			ARDs4StepUpDownMovement[iPull4StepFL].lrZone1Acc						:= fbA31ArmSpeedProfileMemory.ARDsArmSpeedProfileMemory[fbA21UpDownPattern.ARDsUpdownPatternMemory[ARi4StepPatternNo[iPull4StepFL]].iZone1SpdProfileNo].lrAcc;
			ARDs4StepUpDownMovement[iPull4StepFL].lrZone1Dcc						:= fbA31ArmSpeedProfileMemory.ARDsArmSpeedProfileMemory[fbA21UpDownPattern.ARDsUpdownPatternMemory[ARi4StepPatternNo[iPull4StepFL]].iZone1SpdProfileNo].lrDcc;
			ARDs4StepUpDownMovement[iPull4StepFL].lrZone2Acc						:= fbA31ArmSpeedProfileMemory.ARDsArmSpeedProfileMemory[fbA21UpDownPattern.ARDsUpdownPatternMemory[ARi4StepPatternNo[iPull4StepFL]].iZone2SpdProfileNo].lrAcc;
			ARDs4StepUpDownMovement[iPull4StepFL].lrZone2Dcc						:= fbA31ArmSpeedProfileMemory.ARDsArmSpeedProfileMemory[fbA21UpDownPattern.ARDsUpdownPatternMemory[ARi4StepPatternNo[iPull4StepFL]].iZone2SpdProfileNo].lrDcc;
			ARDs4StepUpDownMovement[iPull4StepFL].lrZone3Acc						:= fbA31ArmSpeedProfileMemory.ARDsArmSpeedProfileMemory[fbA21UpDownPattern.ARDsUpdownPatternMemory[ARi4StepPatternNo[iPull4StepFL]].iZone3SpdProfileNo].lrAcc;
			ARDs4StepUpDownMovement[iPull4StepFL].lrZone3Dcc						:= fbA31ArmSpeedProfileMemory.ARDsArmSpeedProfileMemory[fbA21UpDownPattern.ARDsUpdownPatternMemory[ARi4StepPatternNo[iPull4StepFL]].iZone3SpdProfileNo].lrDcc;
			ARDs4StepUpDownMovement[iPull4StepFL].lrZone4Acc						:= fbA31ArmSpeedProfileMemory.ARDsArmSpeedProfileMemory[fbA21UpDownPattern.ARDsUpdownPatternMemory[ARi4StepPatternNo[iPull4StepFL]].iZone4SpdProfileNo].lrAcc;
			ARDs4StepUpDownMovement[iPull4StepFL].lrZone4Dcc						:= fbA31ArmSpeedProfileMemory.ARDsArmSpeedProfileMemory[fbA21UpDownPattern.ARDsUpdownPatternMemory[ARi4StepPatternNo[iPull4StepFL]].iZone4SpdProfileNo].lrDcc;

			ARDs4StepUpDownMovement[iPull4StepFL].sReservedLreal;
			ARDs4StepUpDownMovement[iPull4StepFL].sUpDownPatternDescription	:= fbA21UpDownPattern.ARDsUpdownPatternMemory[ARi4StepPatternNo[iPull4StepFL]].sDescription;
	END_IF
END_FOR

(*[][][][][][][][][][][][][][][][][][][][][][][][][][][][][][][][][][][][][][][][][][][][][][][][][][][][][][][][][][][][][][][][][][][][][][][][][][][][][][][][][][][][][][][][][][][][][][][][][][][]*)
(*Check Which Staton Request for Data*)
iCallCheck := 0;
bCalledDataRequestStationFound := FALSE;

FOR iCallCheck := 0 TO iStnQty DO
		IF ARbProductRecipeCallEn[iCallCheck] THEN
		iCalledDataRequestFromStationNo := iCallCheck;
		bCalledDataRequestStationFound := TRUE;
		iCallCheck := 28;
		END_IF
END_FOR

IF NOT bCalledDataRequestStationFound AND iCallCheck < iStnQty THEN
		iCalledDataRequestFromStationNo := 0;
END_IF

iProductRecipeNoCall := ARiProductRecipeNoCall[iCalledDataRequestFromStationNo];
iProductRecipeStepCall := ARiProductRecipeStepCall[iCalledDataRequestFromStationNo];
bCallSt := bCalledDataRequestStationFound;


(*[][][][][][][][][][][][][][][][][][][][][][][][][][][][][][][][][][][][][][][][][][][][][][][][][][][][][][][][][][][][][][][][][][][][][][][][][][][][][][][][][][][][][][][][][][][][][][][][][][][]*)
(*Reset fb*)
bCallStRE(CLK:=bCallSt , Q=> );
bCallStFE(CLK:=bCallSt , Q=> );

IF bCallStRE.Q OR bCallStFE.Q THEN
DSA1fbPnpSequenceMemoryCall.bCallPB := FALSE;
DSA21UpDownPatternCall.bCallPB := FALSE;
DSA31ArmSpeedProfileCall.bCallPB := FALSE;
DSfbGnrProductRecipeMemoryOut.bCallCompleted := FALSE;
DSfbGnrProductRecipeMemoryOut.bCallArmSpeedProfileMemoryErr := FALSE;
DSfbGnrProductRecipeMemoryOut.bCallUpDownPatternMemoryErr := FALSE;
DSfbGnrProductRecipeMemoryOut.bCallPickStationNoErr := FALSE;
DSfbGnrProductRecipeMemoryOut.bCallTransferStationNoErr := FALSE;

iBufferPickStationNo:= 0;
iBufferTransferStationNo:= 0;
iBufferDownPickPatternNo:= 0;
iBufferUpPickPatternNo:= 0;
iBufferDownTransferPatternNo:= 0;
iBufferUpTransferPatternNo:= 0;
(*
DSfbGnrProductRecipeMemoryOut.DSGnrCalledArmPnpParameter.iCallArmNo := 0;
DSfbGnrProductRecipeMemoryOut.DSGnrCalledArmPnpParameter.iPickStationNo := 0;
DSfbGnrProductRecipeMemoryOut.DSGnrCalledArmPnpParameter.iTransferStationNo := 0;
*)
DSfbGnrProductRecipeMemoryOut.iCallCaseNo := 0;

END_IF
(*
(*Limit Loading and Unloading ID*)
IF ARiLdStnID < iStnQty THEN
ARiLdStnID:= iStnQty + 1;
END_IF
IF ARiUldStnID < iStnQty THEN
ARiUldStnID:= iStnQty + 2;
END_IF
*)


(*Reset Err after 0.5Sec*)
(*
tCallPickStationNoErrTimer(IN:= DSfbGnrProductRecipeMemoryOut.bCallPickStationNoErr , PT:=t#0.5s , Q=> , ET=> );
*)
IF tCallPickStationNoErrTimer.Q OR NOT bCallSt THEN
DSfbGnrProductRecipeMemoryOut.bCallPickStationNoErr := FALSE;
END_IF

(*
tCallTransferStationNoErrTimer(IN:= DSfbGnrProductRecipeMemoryOut.bCallTransferStationNoErr , PT:=t#0.5s , Q=> , ET=> );
*)
IF tCallTransferStationNoErrTimer.Q OR NOT bCallSt THEN
DSfbGnrProductRecipeMemoryOut.bCallTransferStationNoErr := FALSE;
END_IF

(*
tCallArmSpeedProfileMemoryErrTimer(IN:= DSfbGnrProductRecipeMemoryOut.bCallArmSpeedProfileMemoryErr , PT:=t#0.5s , Q=> , ET=> );
*)
IF tCallArmSpeedProfileMemoryErrTimer.Q OR NOT bCallSt THEN
DSfbGnrProductRecipeMemoryOut.bCallArmSpeedProfileMemoryErr := FALSE;
END_IF

(*
tCallUpDownPatternMemoryErrTimer(IN:= DSfbGnrProductRecipeMemoryOut.bCallUpDownPatternMemoryErr , PT:=t#0.5s , Q=> , ET=> );
*)
IF tCallUpDownPatternMemoryErrTimer.Q OR NOT bCallSt THEN
DSfbGnrProductRecipeMemoryOut.bCallUpDownPatternMemoryErr := FALSE;
END_IF

(*Trigger Error*)

IF (iProductRecipeNoCall <= 0 OR iProductRecipeNoCall > iProductRecipeArrayQty) AND bCallSt THEN
DSfbGnrProductRecipeMemoryOut.bInvalidProductRecipeNoErrHold := TRUE;
ELSE
DSfbGnrProductRecipeMemoryOut.bInvalidProductRecipeNoErrHold := FALSE;
END_IF

IF (iProductRecipeStepCall <= 0 OR iProductRecipeStepCall > iProductRecipeStepArrayQty) AND bCallSt THEN
DSfbGnrProductRecipeMemoryOut.bInvalidProductRecipeStepErrHold := TRUE;
ELSE
DSfbGnrProductRecipeMemoryOut.bInvalidProductRecipeStepErrHold := FALSE;
END_IF

rebInvalidProductRecipeNo(CLK:=DSfbGnrProductRecipeMemoryOut.bInvalidProductRecipeNoErrHold AND bCallSt , Q=> );

IF rebInvalidProductRecipeNo.Q THEN
DSfbGnrProductRecipeMemoryOut.bInvalidProductRecipeNoErrPulse := TRUE;
END_IF

rebInvalidProductRecipeStep(CLK:=DSfbGnrProductRecipeMemoryOut.bInvalidProductRecipeStepErrHold AND bCallSt , Q=> );

IF rebInvalidProductRecipeStep.Q THEN
DSfbGnrProductRecipeMemoryOut.bInvalidProductRecipeStepErrPulse := TRUE;
END_IF


tInvalidProductRecipeNoErrTimer(IN:= DSfbGnrProductRecipeMemoryOut.bInvalidProductRecipeNoErrHold , PT:=t#0.5s , Q=> , ET=> );

IF tInvalidProductRecipeNoErrTimer.Q OR NOT bCallSt THEN
DSfbGnrProductRecipeMemoryOut.bInvalidProductRecipeNoErrPulse := FALSE;
END_IF


tInvalidProductRecipeStepErrTimer(IN:= DSfbGnrProductRecipeMemoryOut.bInvalidProductRecipeStepErrHold , PT:=t#0.5s , Q=> , ET=> );

IF tInvalidProductRecipeStepErrTimer.Q OR NOT bCallSt THEN
DSfbGnrProductRecipeMemoryOut.bInvalidProductRecipeStepErrPulse := FALSE;
END_IF

(*Declare FB*)

fbA1PnpSequenceMemory(
	bSavePB:=bSavePB ,
	bLoadPB:= bLoadPB,
	bClearPB:=bClearPB,
	bCopyPB:=DSA1fbPnpSequenceMemoryStore.bCopyPB ,
	iCopyToProductRecipeNo:=DSA1fbPnpSequenceMemoryStore.iCopyToProductRecipeNo ,
(*	ARiLdStnID:= ARiLdStnID,
	ARiUldStnID:= ARiUldStnID,
*)	iProductRecipeNo:=DSA1fbPnpSequenceMemoryStore.iProductRecipeNo ,
	DSA1inPnpSequenceMemory:=DSA1fbPnpSequenceMemoryStore.DsA1inPnpSequenceMemory ,
	Call_iProductRecipeNo:=DSA1fbPnpSequenceMemoryCall.Call_iProductRecipeNo ,
	bCallPB:=DSA1fbPnpSequenceMemoryCall.bCallPB ,
	bSaveInd=>bSaveInd ,
	bLoadInd=> bLoadInd,
	bClearInd=>bClearInd,
	bCallCompleted=>DSA1fbPnpSequenceMemoryCall.bCallCompleted ,
	bInvalidCallProductRecipeNoHold=>DSA1fbPnpSequenceMemoryCall.bInvalidCallProductRecipeNoHold ,
	bInvalidCallProductRecipeNoPulse=>DSA1fbPnpSequenceMemoryCall.bInvalidCallProductRecipeNoPulse ,
	Call_DSA1PnpSequenceMemory=>DSA1fbPnpSequenceMemoryCall.Call_DsPnpSequenceMemory );

fbA21UpDownPattern(
	bSavePB:=bSavePB ,
	bLoadPB:= bLoadPB,
	bCopyPB:=DSA21UpDownPatternStore.bCopyPB ,
	iCopyToUpDownPatternNo:= DSA21UpDownPatternStore.iCopyToUpDownPatternNo,
	iUpDownPatternNo:=DSA21UpDownPatternStore.iUpDownPatternNo ,
	DSinUpDownPatternMemory:=DSA21UpDownPatternStore.DsInUpDownPatternMemory ,
	Call_iUpDownPatternNo:=DSA21UpDownPatternCall.Call_iUpDownPatternNo ,
	bCallPB:=DSA21UpDownPatternCall.bCallPB ,
	bSaveInd=>bSaveInd ,
	bLoadInd=>bLoadInd,
	bCallCompleted=>DSA21UpDownPatternCall.bCallCompleted ,
	bInvalidCallUpdownPatternNoHold=>DSA21UpDownPatternCall.bInvalidCallUpDownPatternNoHold ,
	bInvalidCallUpdownPatternNoPulse=>DSA21UpDownPatternCall.bInvalidCallUpDownPatternNoPulse ,
	Call_DSUpdownPattern=>DSA21UpDownPatternCall.Call_DsUpDownPattern );

fbA31ArmSpeedProfileMemory(
	bSavePB:= bSavePB,
	bLoadPB:= bLoadPB,
	bCopyPB:=DSA31ArmSpeedProfileStore.bCopyPB ,
	iCopyToSpdProfileNo:=DSA31ArmSpeedProfileStore.iCopyToSpdProfileNo ,
	iVertMaxVelo:=iVertMaxVelo ,
	iVertMaxAcc:=iVertMaxAcc ,
	iVertMaxDcc:=iVertMaxDcc ,
	iVertMinVelo:=iVertMinVelo ,
	iVertMinAcc:=iVertMinAcc ,
	iVertMinDcc:=iVertMinDcc ,
	iArmSpdProfileNo:= DSA31ArmSpeedProfileStore.iArmSpdProfileNo,
	DSArmSpeedProfile:= DSA31ArmSpeedProfileStore.DsArmSpeedProfile,
	Call_iArmSpdProfile:= DSA31ArmSpeedProfileCall.Call_iArmSpdProfile ,
	bCallPB:= DSA31ArmSpeedProfileCall.bCallPB ,
	bSaveInd=>bSaveInd ,
	bLoadInd=>bLoadInd ,
	bCallCompleted=>DSA31ArmSpeedProfileCall.bCallCompleted ,
	bInvalidCallArmSpdProfileNoHold=> DSA31ArmSpeedProfileCall.bInvalidCallArmSpdProfileNoHold,
	bInvalidCallArmSpdProfileNoPulse=> DSA31ArmSpeedProfileCall.bInvalidCallArmSpdProfileNoPulse,
	Call_DSArmSpeedProfile=>DSA31ArmSpeedProfileCall.Call_DSArmSpdProfile );

fbV2A32MachineZoneHeight(
	ARDSLdZoneHeight:=ARDSLdZoneHeight ,
	ARDSStationZoneHeight:=ARDSStationZoneHeight ,
	ARDSUldZoneHeight:=ARDSUldZoneHeight ,
	ARDSLdZonePosOut=>ARDSLdZonePosOut ,
	ARDSStationZonePosOut=>ARDSStationZonePosOut ,
	ARDSUldZonePosOut=>ARDSUldZonePosOut );



(*Call Start*)

rebCallSt(CLK:=bCallSt , Q=> );
IF rebCallSt.Q AND NOT DSfbGnrProductRecipeMemoryOut.bInvalidProductRecipeNoErrHold AND NOT DSfbGnrProductRecipeMemoryOut.bInvalidProductRecipeStepErrHold(*) OR febInvalidProcessStep.Q*) THEN
DSfbGnrProductRecipeMemoryOut.iCallCaseNo := 1;
END_IF



rebInvalidUpDownPatternMemoryCall(CLK:=DSA21UpDownPatternCall.bInvalidCallUpDownPatternNoHold , Q=> );
rebInvalidSpeedProfileMemoryCall(CLK:=DSA31ArmSpeedProfileCall.bInvalidCallArmSpdProfileNoHold , Q=> );



CASE DSfbGnrProductRecipeMemoryOut.iCallCaseNo OF

0:;

1: (*Select PnpSequenceNo By Refering iProductRecipeNoCall*)
DSfbGnrProductRecipeMemoryOut.bCallUpDownPatternMemoryErr := FALSE;
DSfbGnrProductRecipeMemoryOut.bCallArmSpeedProfileMemoryErr := FALSE;
DSfbGnrProductRecipeMemoryOut.bCallPickStationNoErr := FALSE;
DSfbGnrProductRecipeMemoryOut.bCallTransferStationNoErr := FALSE;


DSA1fbPnpSequenceMemoryCall.Call_iProductRecipeNo := iProductRecipeNoCall;
DSA1fbPnpSequenceMemoryCall.bCallPB := TRUE;
DSfbGnrProductRecipeMemoryOut.iCalledProductRecipeNo := iProductRecipeNoCall;
DSfbGnrProductRecipeMemoryOut.iCalledProductRecipeStep := iProductRecipeStepCall;

IF DSA1fbPnpSequenceMemoryCall.bCallCompleted THEN
DSA1fbPnpSequenceMemoryCall.bCallPB := FALSE;



DSfbGnrProductRecipeMemoryOut.iCallCaseNo:=10;

END_IF


(*[][][][][][][][][][][][][][][][][][][][][][][][][][][][][][][][][][][][][][][][][][][][][][][][][][][][][][][][][][][][][][][][][][][][][][][][][][][][][][][][][][][][][][][][][][][][][][][][][][][]*)
62: (* Feed Transfer Station Vertical Zone Position*)


DSfbGnrProductRecipeMemoryOut.DSGnrCalledArmPnpParameter.iTransferStationNo := iBufferTransferStationNo;

iTransLdStnID := 0;
iTransUldStnID := 0;
bTransLdStnFound := FALSE;
bTransUldStnFound := FALSE;

iBufTransStnNoCheckFL := 1;
	FOR iBufTransStnNoCheckFL := 1 TO iLdStnQty DO
		IF iBufTransStnNoCheckFL >=1 AND iBufTransStnNoCheckFL <= iLdStnQty THEN
			IF iBufferTransferStationNo = ARiLdStnID[iBufTransStnNoCheckFL] THEN
				iTransLdStnID := iBufTransStnNoCheckFL;
				bTransLdStnFound := TRUE;
				iBufTransStnNoCheckFL := iLdStnQty +2;
			END_IF
		END_IF
	END_FOR

iBufTransStnNoCheckFL := 1;
	FOR iBufTransStnNoCheckFL := 1 TO iUldStnQty DO
		IF iBufTransStnNoCheckFL >=1 AND iBufTransStnNoCheckFL <= iUldStnQty THEN
			IF iBufferTransferStationNo = ARiUldStnID[iBufTransStnNoCheckFL] THEN
				iTransUldStnID := iBufTransStnNoCheckFL;
				bTransUldStnFound := TRUE;
				iBufTransStnNoCheckFL := iUldStnQty +2;
			END_IF
		END_IF
	END_FOR


IF bTransLdStnFound THEN

		IF bEnableCallArmNo THEN
			DSfbGnrProductRecipeMemoryOut.DSGnrCalledArmPnpParameter.DSA1DownTransferMovement.lrZone1StartPos := ARDSLdZonePosOut[iTransLdStnID].lrZone1StartPos - ARiVertArmPosOffset[iCallArmNo] ;
			DSfbGnrProductRecipeMemoryOut.DSGnrCalledArmPnpParameter.DSA1DownTransferMovement.lrZone2StartPos := ARDSLdZonePosOut[iTransLdStnID].lrZone2StartPos - ARiVertArmPosOffset[iCallArmNo] ;
			DSfbGnrProductRecipeMemoryOut.DSGnrCalledArmPnpParameter.DSA1DownTransferMovement.lrZone3StartPos := ARDSLdZonePosOut[iTransLdStnID].lrZone3StartPos - ARiVertArmPosOffset[iCallArmNo] ;
			DSfbGnrProductRecipeMemoryOut.DSGnrCalledArmPnpParameter.DSA1DownTransferMovement.lrZone4StartPos := ARDSLdZonePosOut[iTransLdStnID].lrZone4StartPos - ARiVertArmPosOffset[iCallArmNo] ;

			DSfbGnrProductRecipeMemoryOut.DSGnrCalledArmPnpParameter.DSA1DownTransferMovement.lrZone1EndPos := ARDSLdZonePosOut[iTransLdStnID].lrZone1EndPos - ARiVertArmPosOffset[iCallArmNo] ;
			DSfbGnrProductRecipeMemoryOut.DSGnrCalledArmPnpParameter.DSA1DownTransferMovement.lrZone2EndPos := ARDSLdZonePosOut[iTransLdStnID].lrZone2EndPos - ARiVertArmPosOffset[iCallArmNo] ;
			DSfbGnrProductRecipeMemoryOut.DSGnrCalledArmPnpParameter.DSA1DownTransferMovement.lrZone3EndPos := ARDSLdZonePosOut[iTransLdStnID].lrZone3EndPos - ARiVertArmPosOffset[iCallArmNo] ;
			DSfbGnrProductRecipeMemoryOut.DSGnrCalledArmPnpParameter.DSA1DownTransferMovement.lrZone4EndPos := ARDSLdZonePosOut[iTransLdStnID].lrZone4EndPos - ARiVertArmPosOffset[iCallArmNo] ;

			DSfbGnrProductRecipeMemoryOut.DSGnrCalledArmPnpParameter.DSA1UpTransferMovement.lrZone1StartPos := ARDSLdZonePosOut[iTransLdStnID].lrZone1StartPos - ARiVertArmPosOffset[iCallArmNo] ;
			DSfbGnrProductRecipeMemoryOut.DSGnrCalledArmPnpParameter.DSA1UpTransferMovement.lrZone2StartPos := ARDSLdZonePosOut[iTransLdStnID].lrZone2StartPos - ARiVertArmPosOffset[iCallArmNo] ;
			DSfbGnrProductRecipeMemoryOut.DSGnrCalledArmPnpParameter.DSA1UpTransferMovement.lrZone3StartPos := ARDSLdZonePosOut[iTransLdStnID].lrZone3StartPos - ARiVertArmPosOffset[iCallArmNo] ;
			DSfbGnrProductRecipeMemoryOut.DSGnrCalledArmPnpParameter.DSA1UpTransferMovement.lrZone4StartPos := ARDSLdZonePosOut[iTransLdStnID].lrZone4StartPos - ARiVertArmPosOffset[iCallArmNo] ;

			DSfbGnrProductRecipeMemoryOut.DSGnrCalledArmPnpParameter.DSA1UpTransferMovement.lrZone1EndPos := ARDSLdZonePosOut[iTransLdStnID].lrZone1EndPos - ARiVertArmPosOffset[iCallArmNo] ;
			DSfbGnrProductRecipeMemoryOut.DSGnrCalledArmPnpParameter.DSA1UpTransferMovement.lrZone2EndPos := ARDSLdZonePosOut[iTransLdStnID].lrZone2EndPos - ARiVertArmPosOffset[iCallArmNo] ;
			DSfbGnrProductRecipeMemoryOut.DSGnrCalledArmPnpParameter.DSA1UpTransferMovement.lrZone3EndPos := ARDSLdZonePosOut[iTransLdStnID].lrZone3EndPos - ARiVertArmPosOffset[iCallArmNo] ;
			DSfbGnrProductRecipeMemoryOut.DSGnrCalledArmPnpParameter.DSA1UpTransferMovement.lrZone4EndPos := ARDSLdZonePosOut[iTransLdStnID].lrZone4EndPos - ARiVertArmPosOffset[iCallArmNo] ;

		ELSE

			DSfbGnrProductRecipeMemoryOut.DSGnrCalledArmPnpParameter.DSA1DownTransferMovement.lrZone1StartPos := ARDSLdZonePosOut[iTransLdStnID].lrZone1StartPos - ARiVertArmPosOffset[DSA1fbPnpSequenceMemoryCall.Call_DsPnpSequenceMemory.ARiCallArmNo[iProductRecipeStepCall]] ;
			DSfbGnrProductRecipeMemoryOut.DSGnrCalledArmPnpParameter.DSA1DownTransferMovement.lrZone2StartPos := ARDSLdZonePosOut[iTransLdStnID].lrZone2StartPos - ARiVertArmPosOffset[DSA1fbPnpSequenceMemoryCall.Call_DsPnpSequenceMemory.ARiCallArmNo[iProductRecipeStepCall]] ;
			DSfbGnrProductRecipeMemoryOut.DSGnrCalledArmPnpParameter.DSA1DownTransferMovement.lrZone3StartPos := ARDSLdZonePosOut[iTransLdStnID].lrZone3StartPos - ARiVertArmPosOffset[DSA1fbPnpSequenceMemoryCall.Call_DsPnpSequenceMemory.ARiCallArmNo[iProductRecipeStepCall]] ;
			DSfbGnrProductRecipeMemoryOut.DSGnrCalledArmPnpParameter.DSA1DownTransferMovement.lrZone4StartPos := ARDSLdZonePosOut[iTransLdStnID].lrZone4StartPos - ARiVertArmPosOffset[DSA1fbPnpSequenceMemoryCall.Call_DsPnpSequenceMemory.ARiCallArmNo[iProductRecipeStepCall]] ;

			DSfbGnrProductRecipeMemoryOut.DSGnrCalledArmPnpParameter.DSA1DownTransferMovement.lrZone1EndPos := ARDSLdZonePosOut[iTransLdStnID].lrZone1EndPos - ARiVertArmPosOffset[DSA1fbPnpSequenceMemoryCall.Call_DsPnpSequenceMemory.ARiCallArmNo[iProductRecipeStepCall]] ;
			DSfbGnrProductRecipeMemoryOut.DSGnrCalledArmPnpParameter.DSA1DownTransferMovement.lrZone2EndPos := ARDSLdZonePosOut[iTransLdStnID].lrZone2EndPos - ARiVertArmPosOffset[DSA1fbPnpSequenceMemoryCall.Call_DsPnpSequenceMemory.ARiCallArmNo[iProductRecipeStepCall]] ;
			DSfbGnrProductRecipeMemoryOut.DSGnrCalledArmPnpParameter.DSA1DownTransferMovement.lrZone3EndPos := ARDSLdZonePosOut[iTransLdStnID].lrZone3EndPos - ARiVertArmPosOffset[DSA1fbPnpSequenceMemoryCall.Call_DsPnpSequenceMemory.ARiCallArmNo[iProductRecipeStepCall]] ;
			DSfbGnrProductRecipeMemoryOut.DSGnrCalledArmPnpParameter.DSA1DownTransferMovement.lrZone4EndPos := ARDSLdZonePosOut[iTransLdStnID].lrZone4EndPos - ARiVertArmPosOffset[DSA1fbPnpSequenceMemoryCall.Call_DsPnpSequenceMemory.ARiCallArmNo[iProductRecipeStepCall]];

			DSfbGnrProductRecipeMemoryOut.DSGnrCalledArmPnpParameter.DSA1UpTransferMovement.lrZone1StartPos := ARDSLdZonePosOut[iTransLdStnID].lrZone1StartPos - ARiVertArmPosOffset[DSA1fbPnpSequenceMemoryCall.Call_DsPnpSequenceMemory.ARiCallArmNo[iProductRecipeStepCall]] ;
			DSfbGnrProductRecipeMemoryOut.DSGnrCalledArmPnpParameter.DSA1UpTransferMovement.lrZone2StartPos := ARDSLdZonePosOut[iTransLdStnID].lrZone2StartPos - ARiVertArmPosOffset[DSA1fbPnpSequenceMemoryCall.Call_DsPnpSequenceMemory.ARiCallArmNo[iProductRecipeStepCall]] ;
			DSfbGnrProductRecipeMemoryOut.DSGnrCalledArmPnpParameter.DSA1UpTransferMovement.lrZone3StartPos := ARDSLdZonePosOut[iTransLdStnID].lrZone3StartPos - ARiVertArmPosOffset[DSA1fbPnpSequenceMemoryCall.Call_DsPnpSequenceMemory.ARiCallArmNo[iProductRecipeStepCall]] ;
			DSfbGnrProductRecipeMemoryOut.DSGnrCalledArmPnpParameter.DSA1UpTransferMovement.lrZone4StartPos := ARDSLdZonePosOut[iTransLdStnID].lrZone4StartPos - ARiVertArmPosOffset[DSA1fbPnpSequenceMemoryCall.Call_DsPnpSequenceMemory.ARiCallArmNo[iProductRecipeStepCall]] ;

			DSfbGnrProductRecipeMemoryOut.DSGnrCalledArmPnpParameter.DSA1UpTransferMovement.lrZone1EndPos := ARDSLdZonePosOut[iTransLdStnID].lrZone1EndPos - ARiVertArmPosOffset[DSA1fbPnpSequenceMemoryCall.Call_DsPnpSequenceMemory.ARiCallArmNo[iProductRecipeStepCall]] ;
			DSfbGnrProductRecipeMemoryOut.DSGnrCalledArmPnpParameter.DSA1UpTransferMovement.lrZone2EndPos := ARDSLdZonePosOut[iTransLdStnID].lrZone2EndPos - ARiVertArmPosOffset[DSA1fbPnpSequenceMemoryCall.Call_DsPnpSequenceMemory.ARiCallArmNo[iProductRecipeStepCall]] ;
			DSfbGnrProductRecipeMemoryOut.DSGnrCalledArmPnpParameter.DSA1UpTransferMovement.lrZone3EndPos := ARDSLdZonePosOut[iTransLdStnID].lrZone3EndPos - ARiVertArmPosOffset[DSA1fbPnpSequenceMemoryCall.Call_DsPnpSequenceMemory.ARiCallArmNo[iProductRecipeStepCall]] ;
			DSfbGnrProductRecipeMemoryOut.DSGnrCalledArmPnpParameter.DSA1UpTransferMovement.lrZone4EndPos := ARDSLdZonePosOut[iTransLdStnID].lrZone4EndPos - ARiVertArmPosOffset[DSA1fbPnpSequenceMemoryCall.Call_DsPnpSequenceMemory.ARiCallArmNo[iProductRecipeStepCall]] ;

		END_IF

DSfbGnrProductRecipeMemoryOut.iCallCaseNo:=71;

END_IF


IF bTransUldStnFound THEN

		IF bEnableCallArmNo THEN

			DSfbGnrProductRecipeMemoryOut.DSGnrCalledArmPnpParameter.DSA1DownTransferMovement.lrZone1StartPos := ARDSUldZonePosOut[iTransUldStnID].lrZone1StartPos - ARiVertArmPosOffset[iCallArmNo];
			DSfbGnrProductRecipeMemoryOut.DSGnrCalledArmPnpParameter.DSA1DownTransferMovement.lrZone2StartPos := ARDSUldZonePosOut[iTransUldStnID].lrZone2StartPos - ARiVertArmPosOffset[iCallArmNo];
			DSfbGnrProductRecipeMemoryOut.DSGnrCalledArmPnpParameter.DSA1DownTransferMovement.lrZone3StartPos := ARDSUldZonePosOut[iTransUldStnID].lrZone3StartPos - ARiVertArmPosOffset[iCallArmNo];
			DSfbGnrProductRecipeMemoryOut.DSGnrCalledArmPnpParameter.DSA1DownTransferMovement.lrZone4StartPos := ARDSUldZonePosOut[iTransUldStnID].lrZone4StartPos - ARiVertArmPosOffset[iCallArmNo];

			DSfbGnrProductRecipeMemoryOut.DSGnrCalledArmPnpParameter.DSA1DownTransferMovement.lrZone1EndPos := ARDSUldZonePosOut[iTransUldStnID].lrZone1EndPos - ARiVertArmPosOffset[iCallArmNo];
			DSfbGnrProductRecipeMemoryOut.DSGnrCalledArmPnpParameter.DSA1DownTransferMovement.lrZone2EndPos := ARDSUldZonePosOut[iTransUldStnID].lrZone2EndPos - ARiVertArmPosOffset[iCallArmNo];
			DSfbGnrProductRecipeMemoryOut.DSGnrCalledArmPnpParameter.DSA1DownTransferMovement.lrZone3EndPos := ARDSUldZonePosOut[iTransUldStnID].lrZone3EndPos - ARiVertArmPosOffset[iCallArmNo];
			DSfbGnrProductRecipeMemoryOut.DSGnrCalledArmPnpParameter.DSA1DownTransferMovement.lrZone4EndPos := ARDSUldZonePosOut[iTransUldStnID].lrZone4EndPos - ARiVertArmPosOffset[iCallArmNo];

			DSfbGnrProductRecipeMemoryOut.DSGnrCalledArmPnpParameter.DSA1UpTransferMovement.lrZone1StartPos := ARDSUldZonePosOut[iTransUldStnID].lrZone1StartPos - ARiVertArmPosOffset[iCallArmNo];
			DSfbGnrProductRecipeMemoryOut.DSGnrCalledArmPnpParameter.DSA1UpTransferMovement.lrZone2StartPos := ARDSUldZonePosOut[iTransUldStnID].lrZone2StartPos - ARiVertArmPosOffset[iCallArmNo];
			DSfbGnrProductRecipeMemoryOut.DSGnrCalledArmPnpParameter.DSA1UpTransferMovement.lrZone3StartPos := ARDSUldZonePosOut[iTransUldStnID].lrZone3StartPos - ARiVertArmPosOffset[iCallArmNo];
			DSfbGnrProductRecipeMemoryOut.DSGnrCalledArmPnpParameter.DSA1UpTransferMovement.lrZone4StartPos := ARDSUldZonePosOut[iTransUldStnID].lrZone4StartPos - ARiVertArmPosOffset[iCallArmNo];

			DSfbGnrProductRecipeMemoryOut.DSGnrCalledArmPnpParameter.DSA1UpTransferMovement.lrZone1EndPos := ARDSUldZonePosOut[iTransUldStnID].lrZone1EndPos - ARiVertArmPosOffset[iCallArmNo];
			DSfbGnrProductRecipeMemoryOut.DSGnrCalledArmPnpParameter.DSA1UpTransferMovement.lrZone2EndPos := ARDSUldZonePosOut[iTransUldStnID].lrZone2EndPos - ARiVertArmPosOffset[iCallArmNo];
			DSfbGnrProductRecipeMemoryOut.DSGnrCalledArmPnpParameter.DSA1UpTransferMovement.lrZone3EndPos := ARDSUldZonePosOut[iTransUldStnID].lrZone3EndPos - ARiVertArmPosOffset[iCallArmNo];
			DSfbGnrProductRecipeMemoryOut.DSGnrCalledArmPnpParameter.DSA1UpTransferMovement.lrZone4EndPos := ARDSUldZonePosOut[iTransUldStnID].lrZone4EndPos - ARiVertArmPosOffset[iCallArmNo];

			DSfbGnrProductRecipeMemoryOut.DSGnrCalledArmPnpParameter.DSA1DownTransferMovement.lrMidPos := ARDSUldZonePosOut[iTransUldStnID].lrMidPos;
			DSfbGnrProductRecipeMemoryOut.DSGnrCalledArmPnpParameter.DSA1UpTransferMovement.lrMidPos := ARDSUldZonePosOut[iTransUldStnID].lrMidPos;


		ELSE

			DSfbGnrProductRecipeMemoryOut.DSGnrCalledArmPnpParameter.DSA1DownTransferMovement.lrZone1StartPos := ARDSUldZonePosOut[iTransUldStnID].lrZone1StartPos - ARiVertArmPosOffset[DSA1fbPnpSequenceMemoryCall.Call_DsPnpSequenceMemory.ARiCallArmNo[iProductRecipeStepCall]];
			DSfbGnrProductRecipeMemoryOut.DSGnrCalledArmPnpParameter.DSA1DownTransferMovement.lrZone2StartPos := ARDSUldZonePosOut[iTransUldStnID].lrZone2StartPos - ARiVertArmPosOffset[DSA1fbPnpSequenceMemoryCall.Call_DsPnpSequenceMemory.ARiCallArmNo[iProductRecipeStepCall]];
			DSfbGnrProductRecipeMemoryOut.DSGnrCalledArmPnpParameter.DSA1DownTransferMovement.lrZone3StartPos := ARDSUldZonePosOut[iTransUldStnID].lrZone3StartPos - ARiVertArmPosOffset[DSA1fbPnpSequenceMemoryCall.Call_DsPnpSequenceMemory.ARiCallArmNo[iProductRecipeStepCall]];
			DSfbGnrProductRecipeMemoryOut.DSGnrCalledArmPnpParameter.DSA1DownTransferMovement.lrZone4StartPos := ARDSUldZonePosOut[iTransUldStnID].lrZone4StartPos - ARiVertArmPosOffset[DSA1fbPnpSequenceMemoryCall.Call_DsPnpSequenceMemory.ARiCallArmNo[iProductRecipeStepCall]];

			DSfbGnrProductRecipeMemoryOut.DSGnrCalledArmPnpParameter.DSA1DownTransferMovement.lrZone1EndPos := ARDSUldZonePosOut[iTransUldStnID].lrZone1EndPos - ARiVertArmPosOffset[DSA1fbPnpSequenceMemoryCall.Call_DsPnpSequenceMemory.ARiCallArmNo[iProductRecipeStepCall]];
			DSfbGnrProductRecipeMemoryOut.DSGnrCalledArmPnpParameter.DSA1DownTransferMovement.lrZone2EndPos := ARDSUldZonePosOut[iTransUldStnID].lrZone2EndPos - ARiVertArmPosOffset[DSA1fbPnpSequenceMemoryCall.Call_DsPnpSequenceMemory.ARiCallArmNo[iProductRecipeStepCall]];
			DSfbGnrProductRecipeMemoryOut.DSGnrCalledArmPnpParameter.DSA1DownTransferMovement.lrZone3EndPos := ARDSUldZonePosOut[iTransUldStnID].lrZone3EndPos - ARiVertArmPosOffset[DSA1fbPnpSequenceMemoryCall.Call_DsPnpSequenceMemory.ARiCallArmNo[iProductRecipeStepCall]];
			DSfbGnrProductRecipeMemoryOut.DSGnrCalledArmPnpParameter.DSA1DownTransferMovement.lrZone4EndPos := ARDSUldZonePosOut[iTransUldStnID].lrZone4EndPos - ARiVertArmPosOffset[DSA1fbPnpSequenceMemoryCall.Call_DsPnpSequenceMemory.ARiCallArmNo[iProductRecipeStepCall]];

			DSfbGnrProductRecipeMemoryOut.DSGnrCalledArmPnpParameter.DSA1UpTransferMovement.lrZone1StartPos := ARDSUldZonePosOut[iTransUldStnID].lrZone1StartPos - ARiVertArmPosOffset[DSA1fbPnpSequenceMemoryCall.Call_DsPnpSequenceMemory.ARiCallArmNo[iProductRecipeStepCall]];
			DSfbGnrProductRecipeMemoryOut.DSGnrCalledArmPnpParameter.DSA1UpTransferMovement.lrZone2StartPos := ARDSUldZonePosOut[iTransUldStnID].lrZone2StartPos - ARiVertArmPosOffset[DSA1fbPnpSequenceMemoryCall.Call_DsPnpSequenceMemory.ARiCallArmNo[iProductRecipeStepCall]];
			DSfbGnrProductRecipeMemoryOut.DSGnrCalledArmPnpParameter.DSA1UpTransferMovement.lrZone3StartPos := ARDSUldZonePosOut[iTransUldStnID].lrZone3StartPos - ARiVertArmPosOffset[DSA1fbPnpSequenceMemoryCall.Call_DsPnpSequenceMemory.ARiCallArmNo[iProductRecipeStepCall]];
			DSfbGnrProductRecipeMemoryOut.DSGnrCalledArmPnpParameter.DSA1UpTransferMovement.lrZone4StartPos := ARDSUldZonePosOut[iTransUldStnID].lrZone4StartPos - ARiVertArmPosOffset[DSA1fbPnpSequenceMemoryCall.Call_DsPnpSequenceMemory.ARiCallArmNo[iProductRecipeStepCall]];

			DSfbGnrProductRecipeMemoryOut.DSGnrCalledArmPnpParameter.DSA1UpTransferMovement.lrZone1EndPos := ARDSUldZonePosOut[iTransUldStnID].lrZone1EndPos - ARiVertArmPosOffset[DSA1fbPnpSequenceMemoryCall.Call_DsPnpSequenceMemory.ARiCallArmNo[iProductRecipeStepCall]];
			DSfbGnrProductRecipeMemoryOut.DSGnrCalledArmPnpParameter.DSA1UpTransferMovement.lrZone2EndPos := ARDSUldZonePosOut[iTransUldStnID].lrZone2EndPos - ARiVertArmPosOffset[DSA1fbPnpSequenceMemoryCall.Call_DsPnpSequenceMemory.ARiCallArmNo[iProductRecipeStepCall]];
			DSfbGnrProductRecipeMemoryOut.DSGnrCalledArmPnpParameter.DSA1UpTransferMovement.lrZone3EndPos := ARDSUldZonePosOut[iTransUldStnID].lrZone3EndPos - ARiVertArmPosOffset[DSA1fbPnpSequenceMemoryCall.Call_DsPnpSequenceMemory.ARiCallArmNo[iProductRecipeStepCall]];
			DSfbGnrProductRecipeMemoryOut.DSGnrCalledArmPnpParameter.DSA1UpTransferMovement.lrZone4EndPos := ARDSUldZonePosOut[iTransUldStnID].lrZone4EndPos - ARiVertArmPosOffset[DSA1fbPnpSequenceMemoryCall.Call_DsPnpSequenceMemory.ARiCallArmNo[iProductRecipeStepCall]];

			DSfbGnrProductRecipeMemoryOut.DSGnrCalledArmPnpParameter.DSA1DownTransferMovement.lrMidPos := ARDSUldZonePosOut[iTransUldStnID].lrMidPos;
			DSfbGnrProductRecipeMemoryOut.DSGnrCalledArmPnpParameter.DSA1UpTransferMovement.lrMidPos := ARDSUldZonePosOut[iTransUldStnID].lrMidPos;

		END_IF

DSfbGnrProductRecipeMemoryOut.iCallCaseNo:=71;

END_IF


IF NOT bTransLdStnFound AND NOT bTransUldStnFound AND iBufferTransferStationNo >= 1 AND  iBufferTransferStationNo <= iStnQty THEN

		IF bEnableCallArmNo THEN

			DSfbGnrProductRecipeMemoryOut.DSGnrCalledArmPnpParameter.DSA1DownTransferMovement.lrZone1StartPos := ARDSStationZonePosOut[iBufferTransferStationNo].lrZone1StartPos - ARiVertArmPosOffset[iCallArmNo];
			DSfbGnrProductRecipeMemoryOut.DSGnrCalledArmPnpParameter.DSA1DownTransferMovement.lrZone2StartPos := ARDSStationZonePosOut[iBufferTransferStationNo].lrZone2StartPos - ARiVertArmPosOffset[iCallArmNo];
			DSfbGnrProductRecipeMemoryOut.DSGnrCalledArmPnpParameter.DSA1DownTransferMovement.lrZone3StartPos := ARDSStationZonePosOut[iBufferTransferStationNo].lrZone3StartPos - ARiVertArmPosOffset[iCallArmNo];
			DSfbGnrProductRecipeMemoryOut.DSGnrCalledArmPnpParameter.DSA1DownTransferMovement.lrZone4StartPos := ARDSStationZonePosOut[iBufferTransferStationNo].lrZone4StartPos - ARiVertArmPosOffset[iCallArmNo];

			DSfbGnrProductRecipeMemoryOut.DSGnrCalledArmPnpParameter.DSA1DownTransferMovement.lrZone1EndPos := ARDSStationZonePosOut[iBufferTransferStationNo].lrZone1EndPos - ARiVertArmPosOffset[iCallArmNo];
			DSfbGnrProductRecipeMemoryOut.DSGnrCalledArmPnpParameter.DSA1DownTransferMovement.lrZone2EndPos := ARDSStationZonePosOut[iBufferTransferStationNo].lrZone2EndPos - ARiVertArmPosOffset[iCallArmNo];
			DSfbGnrProductRecipeMemoryOut.DSGnrCalledArmPnpParameter.DSA1DownTransferMovement.lrZone3EndPos := ARDSStationZonePosOut[iBufferTransferStationNo].lrZone3EndPos - ARiVertArmPosOffset[iCallArmNo];
			DSfbGnrProductRecipeMemoryOut.DSGnrCalledArmPnpParameter.DSA1DownTransferMovement.lrZone4EndPos := ARDSStationZonePosOut[iBufferTransferStationNo].lrZone4EndPos - ARiVertArmPosOffset[iCallArmNo];

			DSfbGnrProductRecipeMemoryOut.DSGnrCalledArmPnpParameter.DSA1UpTransferMovement.lrZone1StartPos := ARDSStationZonePosOut[iBufferTransferStationNo].lrZone1StartPos - ARiVertArmPosOffset[iCallArmNo];
			DSfbGnrProductRecipeMemoryOut.DSGnrCalledArmPnpParameter.DSA1UpTransferMovement.lrZone2StartPos := ARDSStationZonePosOut[iBufferTransferStationNo].lrZone2StartPos - ARiVertArmPosOffset[iCallArmNo];
			DSfbGnrProductRecipeMemoryOut.DSGnrCalledArmPnpParameter.DSA1UpTransferMovement.lrZone3StartPos := ARDSStationZonePosOut[iBufferTransferStationNo].lrZone3StartPos - ARiVertArmPosOffset[iCallArmNo];
			DSfbGnrProductRecipeMemoryOut.DSGnrCalledArmPnpParameter.DSA1UpTransferMovement.lrZone4StartPos := ARDSStationZonePosOut[iBufferTransferStationNo].lrZone4StartPos - ARiVertArmPosOffset[iCallArmNo];

			DSfbGnrProductRecipeMemoryOut.DSGnrCalledArmPnpParameter.DSA1UpTransferMovement.lrZone1EndPos := ARDSStationZonePosOut[iBufferTransferStationNo].lrZone1EndPos - ARiVertArmPosOffset[iCallArmNo];
			DSfbGnrProductRecipeMemoryOut.DSGnrCalledArmPnpParameter.DSA1UpTransferMovement.lrZone2EndPos := ARDSStationZonePosOut[iBufferTransferStationNo].lrZone2EndPos - ARiVertArmPosOffset[iCallArmNo];
			DSfbGnrProductRecipeMemoryOut.DSGnrCalledArmPnpParameter.DSA1UpTransferMovement.lrZone3EndPos := ARDSStationZonePosOut[iBufferTransferStationNo].lrZone3EndPos - ARiVertArmPosOffset[iCallArmNo];
			DSfbGnrProductRecipeMemoryOut.DSGnrCalledArmPnpParameter.DSA1UpTransferMovement.lrZone4EndPos := ARDSStationZonePosOut[iBufferTransferStationNo].lrZone4EndPos - ARiVertArmPosOffset[iCallArmNo];

			DSfbGnrProductRecipeMemoryOut.DSGnrCalledArmPnpParameter.DSA1DownTransferMovement.lrMidPos := ARDSStationZonePosOut[iBufferTransferStationNo].lrMidPos;
			DSfbGnrProductRecipeMemoryOut.DSGnrCalledArmPnpParameter.DSA1UpTransferMovement.lrMidPos := ARDSStationZonePosOut[iBufferTransferStationNo].lrMidPos;


		ELSE

			DSfbGnrProductRecipeMemoryOut.DSGnrCalledArmPnpParameter.DSA1DownTransferMovement.lrZone1StartPos := ARDSStationZonePosOut[iBufferTransferStationNo].lrZone1StartPos - ARiVertArmPosOffset[DSA1fbPnpSequenceMemoryCall.Call_DsPnpSequenceMemory.ARiCallArmNo[iProductRecipeStepCall]];
			DSfbGnrProductRecipeMemoryOut.DSGnrCalledArmPnpParameter.DSA1DownTransferMovement.lrZone2StartPos := ARDSStationZonePosOut[iBufferTransferStationNo].lrZone2StartPos - ARiVertArmPosOffset[DSA1fbPnpSequenceMemoryCall.Call_DsPnpSequenceMemory.ARiCallArmNo[iProductRecipeStepCall]];
			DSfbGnrProductRecipeMemoryOut.DSGnrCalledArmPnpParameter.DSA1DownTransferMovement.lrZone3StartPos := ARDSStationZonePosOut[iBufferTransferStationNo].lrZone3StartPos - ARiVertArmPosOffset[DSA1fbPnpSequenceMemoryCall.Call_DsPnpSequenceMemory.ARiCallArmNo[iProductRecipeStepCall]];
			DSfbGnrProductRecipeMemoryOut.DSGnrCalledArmPnpParameter.DSA1DownTransferMovement.lrZone4StartPos := ARDSStationZonePosOut[iBufferTransferStationNo].lrZone4StartPos - ARiVertArmPosOffset[DSA1fbPnpSequenceMemoryCall.Call_DsPnpSequenceMemory.ARiCallArmNo[iProductRecipeStepCall]];

			DSfbGnrProductRecipeMemoryOut.DSGnrCalledArmPnpParameter.DSA1DownTransferMovement.lrZone1EndPos := ARDSStationZonePosOut[iBufferTransferStationNo].lrZone1EndPos - ARiVertArmPosOffset[DSA1fbPnpSequenceMemoryCall.Call_DsPnpSequenceMemory.ARiCallArmNo[iProductRecipeStepCall]];
			DSfbGnrProductRecipeMemoryOut.DSGnrCalledArmPnpParameter.DSA1DownTransferMovement.lrZone2EndPos := ARDSStationZonePosOut[iBufferTransferStationNo].lrZone2EndPos - ARiVertArmPosOffset[DSA1fbPnpSequenceMemoryCall.Call_DsPnpSequenceMemory.ARiCallArmNo[iProductRecipeStepCall]];
			DSfbGnrProductRecipeMemoryOut.DSGnrCalledArmPnpParameter.DSA1DownTransferMovement.lrZone3EndPos := ARDSStationZonePosOut[iBufferTransferStationNo].lrZone3EndPos - ARiVertArmPosOffset[DSA1fbPnpSequenceMemoryCall.Call_DsPnpSequenceMemory.ARiCallArmNo[iProductRecipeStepCall]];
			DSfbGnrProductRecipeMemoryOut.DSGnrCalledArmPnpParameter.DSA1DownTransferMovement.lrZone4EndPos := ARDSStationZonePosOut[iBufferTransferStationNo].lrZone4EndPos - ARiVertArmPosOffset[DSA1fbPnpSequenceMemoryCall.Call_DsPnpSequenceMemory.ARiCallArmNo[iProductRecipeStepCall]];

			DSfbGnrProductRecipeMemoryOut.DSGnrCalledArmPnpParameter.DSA1UpTransferMovement.lrZone1StartPos := ARDSStationZonePosOut[iBufferTransferStationNo].lrZone1StartPos - ARiVertArmPosOffset[DSA1fbPnpSequenceMemoryCall.Call_DsPnpSequenceMemory.ARiCallArmNo[iProductRecipeStepCall]];
			DSfbGnrProductRecipeMemoryOut.DSGnrCalledArmPnpParameter.DSA1UpTransferMovement.lrZone2StartPos := ARDSStationZonePosOut[iBufferTransferStationNo].lrZone2StartPos - ARiVertArmPosOffset[DSA1fbPnpSequenceMemoryCall.Call_DsPnpSequenceMemory.ARiCallArmNo[iProductRecipeStepCall]];
			DSfbGnrProductRecipeMemoryOut.DSGnrCalledArmPnpParameter.DSA1UpTransferMovement.lrZone3StartPos := ARDSStationZonePosOut[iBufferTransferStationNo].lrZone3StartPos - ARiVertArmPosOffset[DSA1fbPnpSequenceMemoryCall.Call_DsPnpSequenceMemory.ARiCallArmNo[iProductRecipeStepCall]];
			DSfbGnrProductRecipeMemoryOut.DSGnrCalledArmPnpParameter.DSA1UpTransferMovement.lrZone4StartPos := ARDSStationZonePosOut[iBufferTransferStationNo].lrZone4StartPos - ARiVertArmPosOffset[DSA1fbPnpSequenceMemoryCall.Call_DsPnpSequenceMemory.ARiCallArmNo[iProductRecipeStepCall]];

			DSfbGnrProductRecipeMemoryOut.DSGnrCalledArmPnpParameter.DSA1UpTransferMovement.lrZone1EndPos := ARDSStationZonePosOut[iBufferTransferStationNo].lrZone1EndPos - ARiVertArmPosOffset[DSA1fbPnpSequenceMemoryCall.Call_DsPnpSequenceMemory.ARiCallArmNo[iProductRecipeStepCall]];
			DSfbGnrProductRecipeMemoryOut.DSGnrCalledArmPnpParameter.DSA1UpTransferMovement.lrZone2EndPos := ARDSStationZonePosOut[iBufferTransferStationNo].lrZone2EndPos - ARiVertArmPosOffset[DSA1fbPnpSequenceMemoryCall.Call_DsPnpSequenceMemory.ARiCallArmNo[iProductRecipeStepCall]];
			DSfbGnrProductRecipeMemoryOut.DSGnrCalledArmPnpParameter.DSA1UpTransferMovement.lrZone3EndPos := ARDSStationZonePosOut[iBufferTransferStationNo].lrZone3EndPos - ARiVertArmPosOffset[DSA1fbPnpSequenceMemoryCall.Call_DsPnpSequenceMemory.ARiCallArmNo[iProductRecipeStepCall]];
			DSfbGnrProductRecipeMemoryOut.DSGnrCalledArmPnpParameter.DSA1UpTransferMovement.lrZone4EndPos := ARDSStationZonePosOut[iBufferTransferStationNo].lrZone4EndPos - ARiVertArmPosOffset[DSA1fbPnpSequenceMemoryCall.Call_DsPnpSequenceMemory.ARiCallArmNo[iProductRecipeStepCall]];

			DSfbGnrProductRecipeMemoryOut.DSGnrCalledArmPnpParameter.DSA1DownTransferMovement.lrMidPos := ARDSStationZonePosOut[iBufferTransferStationNo].lrMidPos;
			DSfbGnrProductRecipeMemoryOut.DSGnrCalledArmPnpParameter.DSA1UpTransferMovement.lrMidPos := ARDSStationZonePosOut[iBufferTransferStationNo].lrMidPos;

		END_IF

DSfbGnrProductRecipeMemoryOut.iCallCaseNo:=71;

END_IF


IF iBufferTransferStationNo < 1 OR (NOT bTransLdStnFound AND NOT bTransUldStnFound AND  iBufferTransferStationNo > iStnQty) THEN

DSfbGnrProductRecipeMemoryOut.iCallCaseNo:=84;
END_IF

61: (* Feed Pick Station Vertical Zone Position*)

DSfbGnrProductRecipeMemoryOut.DSGnrCalledArmPnpParameter.iPickStationNo := iBufferPickStationNo;


iPickLdStnID := 0;
iPickUldStnID := 0;
bPickLdStnFound := FALSE;
bPickUldStnFound := FALSE;

iBufPickStnNoCheckFL := 1;
	FOR iBufPickStnNoCheckFL := 1 TO iLdStnQty DO
		IF iBufPickStnNoCheckFL >=1 AND iBufPickStnNoCheckFL <= iLdStnQty THEN
			IF iBufferPickStationNo = ARiLdStnID[iBufPickStnNoCheckFL] THEN
				iPickLdStnID := iBufPickStnNoCheckFL;
				bPickLdStnFound := TRUE;
				iBufPickStnNoCheckFL := iLdStnQty +2;
			END_IF
		END_IF
	END_FOR

iBufPickStnNoCheckFL := 1;
	FOR iBufPickStnNoCheckFL := 1 TO iUldStnQty DO
		IF iBufPickStnNoCheckFL >=1 AND iBufPickStnNoCheckFL <= iUldStnQty THEN
			IF iBufferPickStationNo = ARiUldStnID[iBufPickStnNoCheckFL] THEN
				iPickUldStnID := iBufPickStnNoCheckFL;
				bPickUldStnFound := TRUE;
				iBufPickStnNoCheckFL := iUldStnQty +2;
			END_IF
		END_IF
	END_FOR


(************************************************)

IF bPickLdStnFound THEN

		IF bEnableCallArmNo THEN

			DSfbGnrProductRecipeMemoryOut.DSGnrCalledArmPnpParameter.DSA1DownPickMovement.lrZone1StartPos := ARDSLdZonePosOut[iPickLdStnID].lrZone1StartPos - ARiVertArmPosOffset[iCallArmNo];
			DSfbGnrProductRecipeMemoryOut.DSGnrCalledArmPnpParameter.DSA1DownPickMovement.lrZone2StartPos := ARDSLdZonePosOut[iPickLdStnID].lrZone2StartPos - ARiVertArmPosOffset[iCallArmNo];
			DSfbGnrProductRecipeMemoryOut.DSGnrCalledArmPnpParameter.DSA1DownPickMovement.lrZone3StartPos := ARDSLdZonePosOut[iPickLdStnID].lrZone3StartPos - ARiVertArmPosOffset[iCallArmNo];
			DSfbGnrProductRecipeMemoryOut.DSGnrCalledArmPnpParameter.DSA1DownPickMovement.lrZone4StartPos := ARDSLdZonePosOut[iPickLdStnID].lrZone4StartPos - ARiVertArmPosOffset[iCallArmNo];

			DSfbGnrProductRecipeMemoryOut.DSGnrCalledArmPnpParameter.DSA1DownPickMovement.lrZone1EndPos := ARDSLdZonePosOut[iPickLdStnID].lrZone1EndPos - ARiVertArmPosOffset[iCallArmNo];
			DSfbGnrProductRecipeMemoryOut.DSGnrCalledArmPnpParameter.DSA1DownPickMovement.lrZone2EndPos := ARDSLdZonePosOut[iPickLdStnID].lrZone2EndPos - ARiVertArmPosOffset[iCallArmNo];
			DSfbGnrProductRecipeMemoryOut.DSGnrCalledArmPnpParameter.DSA1DownPickMovement.lrZone3EndPos := ARDSLdZonePosOut[iPickLdStnID].lrZone3EndPos - ARiVertArmPosOffset[iCallArmNo];
			DSfbGnrProductRecipeMemoryOut.DSGnrCalledArmPnpParameter.DSA1DownPickMovement.lrZone4EndPos := ARDSLdZonePosOut[iPickLdStnID].lrZone4EndPos - ARiVertArmPosOffset[iCallArmNo];

			DSfbGnrProductRecipeMemoryOut.DSGnrCalledArmPnpParameter.DSA1UpPickMovement.lrZone1StartPos := ARDSLdZonePosOut[iPickLdStnID].lrZone1StartPos - ARiVertArmPosOffset[iCallArmNo];
			DSfbGnrProductRecipeMemoryOut.DSGnrCalledArmPnpParameter.DSA1UpPickMovement.lrZone2StartPos := ARDSLdZonePosOut[iPickLdStnID].lrZone2StartPos - ARiVertArmPosOffset[iCallArmNo];
			DSfbGnrProductRecipeMemoryOut.DSGnrCalledArmPnpParameter.DSA1UpPickMovement.lrZone3StartPos := ARDSLdZonePosOut[iPickLdStnID].lrZone3StartPos - ARiVertArmPosOffset[iCallArmNo];
			DSfbGnrProductRecipeMemoryOut.DSGnrCalledArmPnpParameter.DSA1UpPickMovement.lrZone4StartPos := ARDSLdZonePosOut[iPickLdStnID].lrZone4StartPos - ARiVertArmPosOffset[iCallArmNo];

			DSfbGnrProductRecipeMemoryOut.DSGnrCalledArmPnpParameter.DSA1UpPickMovement.lrZone1EndPos := ARDSLdZonePosOut[iPickLdStnID].lrZone1EndPos - ARiVertArmPosOffset[iCallArmNo];
			DSfbGnrProductRecipeMemoryOut.DSGnrCalledArmPnpParameter.DSA1UpPickMovement.lrZone2EndPos := ARDSLdZonePosOut[iPickLdStnID].lrZone2EndPos - ARiVertArmPosOffset[iCallArmNo];
			DSfbGnrProductRecipeMemoryOut.DSGnrCalledArmPnpParameter.DSA1UpPickMovement.lrZone3EndPos := ARDSLdZonePosOut[iPickLdStnID].lrZone3EndPos - ARiVertArmPosOffset[iCallArmNo];
			DSfbGnrProductRecipeMemoryOut.DSGnrCalledArmPnpParameter.DSA1UpPickMovement.lrZone4EndPos := ARDSLdZonePosOut[iPickLdStnID].lrZone4EndPos - ARiVertArmPosOffset[iCallArmNo];

			DSfbGnrProductRecipeMemoryOut.DSGnrCalledArmPnpParameter.DSA1DownPickMovement.lrMidPos := ARDSLdZonePosOut[iPickLdStnID].lrMidPos;
			DSfbGnrProductRecipeMemoryOut.DSGnrCalledArmPnpParameter.DSA1UpPickMovement.lrMidPos := ARDSLdZonePosOut[iPickLdStnID].lrMidPos;

		ELSE

			DSfbGnrProductRecipeMemoryOut.DSGnrCalledArmPnpParameter.DSA1DownPickMovement.lrZone1StartPos := ARDSLdZonePosOut[iPickLdStnID].lrZone1StartPos - ARiVertArmPosOffset[DSA1fbPnpSequenceMemoryCall.Call_DsPnpSequenceMemory.ARiCallArmNo[iProductRecipeStepCall]];
			DSfbGnrProductRecipeMemoryOut.DSGnrCalledArmPnpParameter.DSA1DownPickMovement.lrZone2StartPos := ARDSLdZonePosOut[iPickLdStnID].lrZone2StartPos - ARiVertArmPosOffset[DSA1fbPnpSequenceMemoryCall.Call_DsPnpSequenceMemory.ARiCallArmNo[iProductRecipeStepCall]];
			DSfbGnrProductRecipeMemoryOut.DSGnrCalledArmPnpParameter.DSA1DownPickMovement.lrZone3StartPos := ARDSLdZonePosOut[iPickLdStnID].lrZone3StartPos - ARiVertArmPosOffset[DSA1fbPnpSequenceMemoryCall.Call_DsPnpSequenceMemory.ARiCallArmNo[iProductRecipeStepCall]];
			DSfbGnrProductRecipeMemoryOut.DSGnrCalledArmPnpParameter.DSA1DownPickMovement.lrZone4StartPos := ARDSLdZonePosOut[iPickLdStnID].lrZone4StartPos - ARiVertArmPosOffset[DSA1fbPnpSequenceMemoryCall.Call_DsPnpSequenceMemory.ARiCallArmNo[iProductRecipeStepCall]];

			DSfbGnrProductRecipeMemoryOut.DSGnrCalledArmPnpParameter.DSA1DownPickMovement.lrZone1EndPos := ARDSLdZonePosOut[iPickLdStnID].lrZone1EndPos - ARiVertArmPosOffset[DSA1fbPnpSequenceMemoryCall.Call_DsPnpSequenceMemory.ARiCallArmNo[iProductRecipeStepCall]];
			DSfbGnrProductRecipeMemoryOut.DSGnrCalledArmPnpParameter.DSA1DownPickMovement.lrZone2EndPos := ARDSLdZonePosOut[iPickLdStnID].lrZone2EndPos - ARiVertArmPosOffset[DSA1fbPnpSequenceMemoryCall.Call_DsPnpSequenceMemory.ARiCallArmNo[iProductRecipeStepCall]];
			DSfbGnrProductRecipeMemoryOut.DSGnrCalledArmPnpParameter.DSA1DownPickMovement.lrZone3EndPos := ARDSLdZonePosOut[iPickLdStnID].lrZone3EndPos - ARiVertArmPosOffset[DSA1fbPnpSequenceMemoryCall.Call_DsPnpSequenceMemory.ARiCallArmNo[iProductRecipeStepCall]];
			DSfbGnrProductRecipeMemoryOut.DSGnrCalledArmPnpParameter.DSA1DownPickMovement.lrZone4EndPos := ARDSLdZonePosOut[iPickLdStnID].lrZone4EndPos - ARiVertArmPosOffset[DSA1fbPnpSequenceMemoryCall.Call_DsPnpSequenceMemory.ARiCallArmNo[iProductRecipeStepCall]];

			DSfbGnrProductRecipeMemoryOut.DSGnrCalledArmPnpParameter.DSA1UpPickMovement.lrZone1StartPos := ARDSLdZonePosOut[iPickLdStnID].lrZone1StartPos - ARiVertArmPosOffset[DSA1fbPnpSequenceMemoryCall.Call_DsPnpSequenceMemory.ARiCallArmNo[iProductRecipeStepCall]];
			DSfbGnrProductRecipeMemoryOut.DSGnrCalledArmPnpParameter.DSA1UpPickMovement.lrZone2StartPos := ARDSLdZonePosOut[iPickLdStnID].lrZone2StartPos - ARiVertArmPosOffset[DSA1fbPnpSequenceMemoryCall.Call_DsPnpSequenceMemory.ARiCallArmNo[iProductRecipeStepCall]];
			DSfbGnrProductRecipeMemoryOut.DSGnrCalledArmPnpParameter.DSA1UpPickMovement.lrZone3StartPos := ARDSLdZonePosOut[iPickLdStnID].lrZone3StartPos - ARiVertArmPosOffset[DSA1fbPnpSequenceMemoryCall.Call_DsPnpSequenceMemory.ARiCallArmNo[iProductRecipeStepCall]];
			DSfbGnrProductRecipeMemoryOut.DSGnrCalledArmPnpParameter.DSA1UpPickMovement.lrZone4StartPos := ARDSLdZonePosOut[iPickLdStnID].lrZone4StartPos - ARiVertArmPosOffset[DSA1fbPnpSequenceMemoryCall.Call_DsPnpSequenceMemory.ARiCallArmNo[iProductRecipeStepCall]];

			DSfbGnrProductRecipeMemoryOut.DSGnrCalledArmPnpParameter.DSA1UpPickMovement.lrZone1EndPos := ARDSLdZonePosOut[iPickLdStnID].lrZone1EndPos - ARiVertArmPosOffset[DSA1fbPnpSequenceMemoryCall.Call_DsPnpSequenceMemory.ARiCallArmNo[iProductRecipeStepCall]];
			DSfbGnrProductRecipeMemoryOut.DSGnrCalledArmPnpParameter.DSA1UpPickMovement.lrZone2EndPos := ARDSLdZonePosOut[iPickLdStnID].lrZone2EndPos - ARiVertArmPosOffset[DSA1fbPnpSequenceMemoryCall.Call_DsPnpSequenceMemory.ARiCallArmNo[iProductRecipeStepCall]];
			DSfbGnrProductRecipeMemoryOut.DSGnrCalledArmPnpParameter.DSA1UpPickMovement.lrZone3EndPos := ARDSLdZonePosOut[iPickLdStnID].lrZone3EndPos - ARiVertArmPosOffset[DSA1fbPnpSequenceMemoryCall.Call_DsPnpSequenceMemory.ARiCallArmNo[iProductRecipeStepCall]];
			DSfbGnrProductRecipeMemoryOut.DSGnrCalledArmPnpParameter.DSA1UpPickMovement.lrZone4EndPos := ARDSLdZonePosOut[iPickLdStnID].lrZone4EndPos - ARiVertArmPosOffset[DSA1fbPnpSequenceMemoryCall.Call_DsPnpSequenceMemory.ARiCallArmNo[iProductRecipeStepCall]];

			DSfbGnrProductRecipeMemoryOut.DSGnrCalledArmPnpParameter.DSA1DownPickMovement.lrMidPos := ARDSLdZonePosOut[iPickLdStnID].lrMidPos;
			DSfbGnrProductRecipeMemoryOut.DSGnrCalledArmPnpParameter.DSA1UpPickMovement.lrMidPos := ARDSLdZonePosOut[iPickLdStnID].lrMidPos;

		END_IF

DSfbGnrProductRecipeMemoryOut.iCallCaseNo:=62;

END_IF


IF bPickUldStnFound THEN

		IF bEnableCallArmNo THEN

			DSfbGnrProductRecipeMemoryOut.DSGnrCalledArmPnpParameter.DSA1DownPickMovement.lrZone1StartPos := ARDSUldZonePosOut[iPickUldStnID].lrZone1StartPos - ARiVertArmPosOffset[iCallArmNo];
			DSfbGnrProductRecipeMemoryOut.DSGnrCalledArmPnpParameter.DSA1DownPickMovement.lrZone2StartPos := ARDSUldZonePosOut[iPickUldStnID].lrZone2StartPos - ARiVertArmPosOffset[iCallArmNo];
			DSfbGnrProductRecipeMemoryOut.DSGnrCalledArmPnpParameter.DSA1DownPickMovement.lrZone3StartPos := ARDSUldZonePosOut[iPickUldStnID].lrZone3StartPos - ARiVertArmPosOffset[iCallArmNo];
			DSfbGnrProductRecipeMemoryOut.DSGnrCalledArmPnpParameter.DSA1DownPickMovement.lrZone4StartPos := ARDSUldZonePosOut[iPickUldStnID].lrZone4StartPos - ARiVertArmPosOffset[iCallArmNo];

			DSfbGnrProductRecipeMemoryOut.DSGnrCalledArmPnpParameter.DSA1DownPickMovement.lrZone1EndPos := ARDSUldZonePosOut[iPickUldStnID].lrZone1EndPos - ARiVertArmPosOffset[iCallArmNo];
			DSfbGnrProductRecipeMemoryOut.DSGnrCalledArmPnpParameter.DSA1DownPickMovement.lrZone2EndPos := ARDSUldZonePosOut[iPickUldStnID].lrZone2EndPos - ARiVertArmPosOffset[iCallArmNo];
			DSfbGnrProductRecipeMemoryOut.DSGnrCalledArmPnpParameter.DSA1DownPickMovement.lrZone3EndPos := ARDSUldZonePosOut[iPickUldStnID].lrZone3EndPos - ARiVertArmPosOffset[iCallArmNo];
			DSfbGnrProductRecipeMemoryOut.DSGnrCalledArmPnpParameter.DSA1DownPickMovement.lrZone4EndPos := ARDSUldZonePosOut[iPickUldStnID].lrZone4EndPos - ARiVertArmPosOffset[iCallArmNo];

			DSfbGnrProductRecipeMemoryOut.DSGnrCalledArmPnpParameter.DSA1UpPickMovement.lrZone1StartPos := ARDSUldZonePosOut[iPickUldStnID].lrZone1StartPos - ARiVertArmPosOffset[iCallArmNo];
			DSfbGnrProductRecipeMemoryOut.DSGnrCalledArmPnpParameter.DSA1UpPickMovement.lrZone2StartPos := ARDSUldZonePosOut[iPickUldStnID].lrZone2StartPos - ARiVertArmPosOffset[iCallArmNo];
			DSfbGnrProductRecipeMemoryOut.DSGnrCalledArmPnpParameter.DSA1UpPickMovement.lrZone3StartPos := ARDSUldZonePosOut[iPickUldStnID].lrZone3StartPos - ARiVertArmPosOffset[iCallArmNo];
			DSfbGnrProductRecipeMemoryOut.DSGnrCalledArmPnpParameter.DSA1UpPickMovement.lrZone4StartPos := ARDSUldZonePosOut[iPickUldStnID].lrZone4StartPos - ARiVertArmPosOffset[iCallArmNo];

			DSfbGnrProductRecipeMemoryOut.DSGnrCalledArmPnpParameter.DSA1UpPickMovement.lrZone1EndPos := ARDSUldZonePosOut[iPickUldStnID].lrZone1EndPos - ARiVertArmPosOffset[iCallArmNo];
			DSfbGnrProductRecipeMemoryOut.DSGnrCalledArmPnpParameter.DSA1UpPickMovement.lrZone2EndPos := ARDSUldZonePosOut[iPickUldStnID].lrZone2EndPos - ARiVertArmPosOffset[iCallArmNo];
			DSfbGnrProductRecipeMemoryOut.DSGnrCalledArmPnpParameter.DSA1UpPickMovement.lrZone3EndPos := ARDSUldZonePosOut[iPickUldStnID].lrZone3EndPos - ARiVertArmPosOffset[iCallArmNo];
			DSfbGnrProductRecipeMemoryOut.DSGnrCalledArmPnpParameter.DSA1UpPickMovement.lrZone4EndPos := ARDSUldZonePosOut[iPickUldStnID].lrZone4EndPos - ARiVertArmPosOffset[iCallArmNo];

			DSfbGnrProductRecipeMemoryOut.DSGnrCalledArmPnpParameter.DSA1DownPickMovement.lrMidPos := ARDSUldZonePosOut[iPickUldStnID].lrMidPos;
			DSfbGnrProductRecipeMemoryOut.DSGnrCalledArmPnpParameter.DSA1UpPickMovement.lrMidPos := ARDSUldZonePosOut[iPickUldStnID].lrMidPos;

		ELSE

			DSfbGnrProductRecipeMemoryOut.DSGnrCalledArmPnpParameter.DSA1DownPickMovement.lrZone1StartPos := ARDSUldZonePosOut[iPickUldStnID].lrZone1StartPos - ARiVertArmPosOffset[DSA1fbPnpSequenceMemoryCall.Call_DsPnpSequenceMemory.ARiCallArmNo[iProductRecipeStepCall]];
			DSfbGnrProductRecipeMemoryOut.DSGnrCalledArmPnpParameter.DSA1DownPickMovement.lrZone2StartPos := ARDSUldZonePosOut[iPickUldStnID].lrZone2StartPos - ARiVertArmPosOffset[DSA1fbPnpSequenceMemoryCall.Call_DsPnpSequenceMemory.ARiCallArmNo[iProductRecipeStepCall]];
			DSfbGnrProductRecipeMemoryOut.DSGnrCalledArmPnpParameter.DSA1DownPickMovement.lrZone3StartPos := ARDSUldZonePosOut[iPickUldStnID].lrZone3StartPos - ARiVertArmPosOffset[DSA1fbPnpSequenceMemoryCall.Call_DsPnpSequenceMemory.ARiCallArmNo[iProductRecipeStepCall]];
			DSfbGnrProductRecipeMemoryOut.DSGnrCalledArmPnpParameter.DSA1DownPickMovement.lrZone4StartPos := ARDSUldZonePosOut[iPickUldStnID].lrZone4StartPos - ARiVertArmPosOffset[DSA1fbPnpSequenceMemoryCall.Call_DsPnpSequenceMemory.ARiCallArmNo[iProductRecipeStepCall]];

			DSfbGnrProductRecipeMemoryOut.DSGnrCalledArmPnpParameter.DSA1DownPickMovement.lrZone1EndPos := ARDSUldZonePosOut[iPickUldStnID].lrZone1EndPos - ARiVertArmPosOffset[DSA1fbPnpSequenceMemoryCall.Call_DsPnpSequenceMemory.ARiCallArmNo[iProductRecipeStepCall]];
			DSfbGnrProductRecipeMemoryOut.DSGnrCalledArmPnpParameter.DSA1DownPickMovement.lrZone2EndPos := ARDSUldZonePosOut[iPickUldStnID].lrZone2EndPos - ARiVertArmPosOffset[DSA1fbPnpSequenceMemoryCall.Call_DsPnpSequenceMemory.ARiCallArmNo[iProductRecipeStepCall]];
			DSfbGnrProductRecipeMemoryOut.DSGnrCalledArmPnpParameter.DSA1DownPickMovement.lrZone3EndPos := ARDSUldZonePosOut[iPickUldStnID].lrZone3EndPos - ARiVertArmPosOffset[DSA1fbPnpSequenceMemoryCall.Call_DsPnpSequenceMemory.ARiCallArmNo[iProductRecipeStepCall]];
			DSfbGnrProductRecipeMemoryOut.DSGnrCalledArmPnpParameter.DSA1DownPickMovement.lrZone4EndPos := ARDSUldZonePosOut[iPickUldStnID].lrZone4EndPos - ARiVertArmPosOffset[DSA1fbPnpSequenceMemoryCall.Call_DsPnpSequenceMemory.ARiCallArmNo[iProductRecipeStepCall]];

			DSfbGnrProductRecipeMemoryOut.DSGnrCalledArmPnpParameter.DSA1UpPickMovement.lrZone1StartPos := ARDSUldZonePosOut[iPickUldStnID].lrZone1StartPos - ARiVertArmPosOffset[DSA1fbPnpSequenceMemoryCall.Call_DsPnpSequenceMemory.ARiCallArmNo[iProductRecipeStepCall]];
			DSfbGnrProductRecipeMemoryOut.DSGnrCalledArmPnpParameter.DSA1UpPickMovement.lrZone2StartPos := ARDSUldZonePosOut[iPickUldStnID].lrZone2StartPos - ARiVertArmPosOffset[DSA1fbPnpSequenceMemoryCall.Call_DsPnpSequenceMemory.ARiCallArmNo[iProductRecipeStepCall]];
			DSfbGnrProductRecipeMemoryOut.DSGnrCalledArmPnpParameter.DSA1UpPickMovement.lrZone3StartPos := ARDSUldZonePosOut[iPickUldStnID].lrZone3StartPos - ARiVertArmPosOffset[DSA1fbPnpSequenceMemoryCall.Call_DsPnpSequenceMemory.ARiCallArmNo[iProductRecipeStepCall]];
			DSfbGnrProductRecipeMemoryOut.DSGnrCalledArmPnpParameter.DSA1UpPickMovement.lrZone4StartPos := ARDSUldZonePosOut[iPickUldStnID].lrZone4StartPos - ARiVertArmPosOffset[DSA1fbPnpSequenceMemoryCall.Call_DsPnpSequenceMemory.ARiCallArmNo[iProductRecipeStepCall]];

			DSfbGnrProductRecipeMemoryOut.DSGnrCalledArmPnpParameter.DSA1UpPickMovement.lrZone1EndPos := ARDSUldZonePosOut[iPickUldStnID].lrZone1EndPos - ARiVertArmPosOffset[DSA1fbPnpSequenceMemoryCall.Call_DsPnpSequenceMemory.ARiCallArmNo[iProductRecipeStepCall]];
			DSfbGnrProductRecipeMemoryOut.DSGnrCalledArmPnpParameter.DSA1UpPickMovement.lrZone2EndPos := ARDSUldZonePosOut[iPickUldStnID].lrZone2EndPos - ARiVertArmPosOffset[DSA1fbPnpSequenceMemoryCall.Call_DsPnpSequenceMemory.ARiCallArmNo[iProductRecipeStepCall]];
			DSfbGnrProductRecipeMemoryOut.DSGnrCalledArmPnpParameter.DSA1UpPickMovement.lrZone3EndPos := ARDSUldZonePosOut[iPickUldStnID].lrZone3EndPos - ARiVertArmPosOffset[DSA1fbPnpSequenceMemoryCall.Call_DsPnpSequenceMemory.ARiCallArmNo[iProductRecipeStepCall]];
			DSfbGnrProductRecipeMemoryOut.DSGnrCalledArmPnpParameter.DSA1UpPickMovement.lrZone4EndPos := ARDSUldZonePosOut[iPickUldStnID].lrZone4EndPos - ARiVertArmPosOffset[DSA1fbPnpSequenceMemoryCall.Call_DsPnpSequenceMemory.ARiCallArmNo[iProductRecipeStepCall]];

			DSfbGnrProductRecipeMemoryOut.DSGnrCalledArmPnpParameter.DSA1DownPickMovement.lrMidPos := ARDSUldZonePosOut[iPickUldStnID].lrMidPos;
			DSfbGnrProductRecipeMemoryOut.DSGnrCalledArmPnpParameter.DSA1UpPickMovement.lrMidPos := ARDSUldZonePosOut[iPickUldStnID].lrMidPos;

END_IF

DSfbGnrProductRecipeMemoryOut.iCallCaseNo:=62;

END_IF


IF NOT bPickLdStnFound AND NOT bPickUldStnFound AND iBufferPickStationNo >= 1 AND  iBufferPickStationNo <= iStnQty THEN

		IF bEnableCallArmNo THEN

			DSfbGnrProductRecipeMemoryOut.DSGnrCalledArmPnpParameter.DSA1DownPickMovement.lrZone1StartPos := ARDSStationZonePosOut[iBufferPickStationNo].lrZone1StartPos - ARiVertArmPosOffset[iCallArmNo];
			DSfbGnrProductRecipeMemoryOut.DSGnrCalledArmPnpParameter.DSA1DownPickMovement.lrZone2StartPos := ARDSStationZonePosOut[iBufferPickStationNo].lrZone2StartPos - ARiVertArmPosOffset[iCallArmNo];
			DSfbGnrProductRecipeMemoryOut.DSGnrCalledArmPnpParameter.DSA1DownPickMovement.lrZone3StartPos := ARDSStationZonePosOut[iBufferPickStationNo].lrZone3StartPos - ARiVertArmPosOffset[iCallArmNo];
			DSfbGnrProductRecipeMemoryOut.DSGnrCalledArmPnpParameter.DSA1DownPickMovement.lrZone4StartPos := ARDSStationZonePosOut[iBufferPickStationNo].lrZone4StartPos - ARiVertArmPosOffset[iCallArmNo];

			DSfbGnrProductRecipeMemoryOut.DSGnrCalledArmPnpParameter.DSA1DownPickMovement.lrZone1EndPos := ARDSStationZonePosOut[iBufferPickStationNo].lrZone1EndPos - ARiVertArmPosOffset[iCallArmNo];
			DSfbGnrProductRecipeMemoryOut.DSGnrCalledArmPnpParameter.DSA1DownPickMovement.lrZone2EndPos := ARDSStationZonePosOut[iBufferPickStationNo].lrZone2EndPos - ARiVertArmPosOffset[iCallArmNo];
			DSfbGnrProductRecipeMemoryOut.DSGnrCalledArmPnpParameter.DSA1DownPickMovement.lrZone3EndPos := ARDSStationZonePosOut[iBufferPickStationNo].lrZone3EndPos - ARiVertArmPosOffset[iCallArmNo];
			DSfbGnrProductRecipeMemoryOut.DSGnrCalledArmPnpParameter.DSA1DownPickMovement.lrZone4EndPos := ARDSStationZonePosOut[iBufferPickStationNo].lrZone4EndPos - ARiVertArmPosOffset[iCallArmNo];

			DSfbGnrProductRecipeMemoryOut.DSGnrCalledArmPnpParameter.DSA1UpPickMovement.lrZone1StartPos := ARDSStationZonePosOut[iBufferPickStationNo].lrZone1StartPos - ARiVertArmPosOffset[iCallArmNo];
			DSfbGnrProductRecipeMemoryOut.DSGnrCalledArmPnpParameter.DSA1UpPickMovement.lrZone2StartPos := ARDSStationZonePosOut[iBufferPickStationNo].lrZone2StartPos - ARiVertArmPosOffset[iCallArmNo];
			DSfbGnrProductRecipeMemoryOut.DSGnrCalledArmPnpParameter.DSA1UpPickMovement.lrZone3StartPos := ARDSStationZonePosOut[iBufferPickStationNo].lrZone3StartPos - ARiVertArmPosOffset[iCallArmNo];
			DSfbGnrProductRecipeMemoryOut.DSGnrCalledArmPnpParameter.DSA1UpPickMovement.lrZone4StartPos := ARDSStationZonePosOut[iBufferPickStationNo].lrZone4StartPos - ARiVertArmPosOffset[iCallArmNo];

			DSfbGnrProductRecipeMemoryOut.DSGnrCalledArmPnpParameter.DSA1UpPickMovement.lrZone1EndPos := ARDSStationZonePosOut[iBufferPickStationNo].lrZone1EndPos - ARiVertArmPosOffset[iCallArmNo];
			DSfbGnrProductRecipeMemoryOut.DSGnrCalledArmPnpParameter.DSA1UpPickMovement.lrZone2EndPos := ARDSStationZonePosOut[iBufferPickStationNo].lrZone2EndPos - ARiVertArmPosOffset[iCallArmNo];
			DSfbGnrProductRecipeMemoryOut.DSGnrCalledArmPnpParameter.DSA1UpPickMovement.lrZone3EndPos := ARDSStationZonePosOut[iBufferPickStationNo].lrZone3EndPos - ARiVertArmPosOffset[iCallArmNo];
			DSfbGnrProductRecipeMemoryOut.DSGnrCalledArmPnpParameter.DSA1UpPickMovement.lrZone4EndPos := ARDSStationZonePosOut[iBufferPickStationNo].lrZone4EndPos - ARiVertArmPosOffset[iCallArmNo];

			DSfbGnrProductRecipeMemoryOut.DSGnrCalledArmPnpParameter.DSA1DownPickMovement.lrMidPos := ARDSStationZonePosOut[iBufferPickStationNo].lrMidPos;
			DSfbGnrProductRecipeMemoryOut.DSGnrCalledArmPnpParameter.DSA1UpPickMovement.lrMidPos := ARDSStationZonePosOut[iBufferPickStationNo].lrMidPos;

		ELSE

			DSfbGnrProductRecipeMemoryOut.DSGnrCalledArmPnpParameter.DSA1DownPickMovement.lrZone1StartPos := ARDSStationZonePosOut[iBufferPickStationNo].lrZone1StartPos - ARiVertArmPosOffset[DSA1fbPnpSequenceMemoryCall.Call_DsPnpSequenceMemory.ARiCallArmNo[iProductRecipeStepCall]];
			DSfbGnrProductRecipeMemoryOut.DSGnrCalledArmPnpParameter.DSA1DownPickMovement.lrZone2StartPos := ARDSStationZonePosOut[iBufferPickStationNo].lrZone2StartPos - ARiVertArmPosOffset[DSA1fbPnpSequenceMemoryCall.Call_DsPnpSequenceMemory.ARiCallArmNo[iProductRecipeStepCall]];
			DSfbGnrProductRecipeMemoryOut.DSGnrCalledArmPnpParameter.DSA1DownPickMovement.lrZone3StartPos := ARDSStationZonePosOut[iBufferPickStationNo].lrZone3StartPos - ARiVertArmPosOffset[DSA1fbPnpSequenceMemoryCall.Call_DsPnpSequenceMemory.ARiCallArmNo[iProductRecipeStepCall]];
			DSfbGnrProductRecipeMemoryOut.DSGnrCalledArmPnpParameter.DSA1DownPickMovement.lrZone4StartPos := ARDSStationZonePosOut[iBufferPickStationNo].lrZone4StartPos - ARiVertArmPosOffset[DSA1fbPnpSequenceMemoryCall.Call_DsPnpSequenceMemory.ARiCallArmNo[iProductRecipeStepCall]];

			DSfbGnrProductRecipeMemoryOut.DSGnrCalledArmPnpParameter.DSA1DownPickMovement.lrZone1EndPos := ARDSStationZonePosOut[iBufferPickStationNo].lrZone1EndPos - ARiVertArmPosOffset[DSA1fbPnpSequenceMemoryCall.Call_DsPnpSequenceMemory.ARiCallArmNo[iProductRecipeStepCall]];
			DSfbGnrProductRecipeMemoryOut.DSGnrCalledArmPnpParameter.DSA1DownPickMovement.lrZone2EndPos := ARDSStationZonePosOut[iBufferPickStationNo].lrZone2EndPos - ARiVertArmPosOffset[DSA1fbPnpSequenceMemoryCall.Call_DsPnpSequenceMemory.ARiCallArmNo[iProductRecipeStepCall]];
			DSfbGnrProductRecipeMemoryOut.DSGnrCalledArmPnpParameter.DSA1DownPickMovement.lrZone3EndPos := ARDSStationZonePosOut[iBufferPickStationNo].lrZone3EndPos - ARiVertArmPosOffset[DSA1fbPnpSequenceMemoryCall.Call_DsPnpSequenceMemory.ARiCallArmNo[iProductRecipeStepCall]];
			DSfbGnrProductRecipeMemoryOut.DSGnrCalledArmPnpParameter.DSA1DownPickMovement.lrZone4EndPos := ARDSStationZonePosOut[iBufferPickStationNo].lrZone4EndPos - ARiVertArmPosOffset[DSA1fbPnpSequenceMemoryCall.Call_DsPnpSequenceMemory.ARiCallArmNo[iProductRecipeStepCall]];

			DSfbGnrProductRecipeMemoryOut.DSGnrCalledArmPnpParameter.DSA1UpPickMovement.lrZone1StartPos := ARDSStationZonePosOut[iBufferPickStationNo].lrZone1StartPos - ARiVertArmPosOffset[DSA1fbPnpSequenceMemoryCall.Call_DsPnpSequenceMemory.ARiCallArmNo[iProductRecipeStepCall]];
			DSfbGnrProductRecipeMemoryOut.DSGnrCalledArmPnpParameter.DSA1UpPickMovement.lrZone2StartPos := ARDSStationZonePosOut[iBufferPickStationNo].lrZone2StartPos - ARiVertArmPosOffset[DSA1fbPnpSequenceMemoryCall.Call_DsPnpSequenceMemory.ARiCallArmNo[iProductRecipeStepCall]];
			DSfbGnrProductRecipeMemoryOut.DSGnrCalledArmPnpParameter.DSA1UpPickMovement.lrZone3StartPos := ARDSStationZonePosOut[iBufferPickStationNo].lrZone3StartPos - ARiVertArmPosOffset[DSA1fbPnpSequenceMemoryCall.Call_DsPnpSequenceMemory.ARiCallArmNo[iProductRecipeStepCall]];
			DSfbGnrProductRecipeMemoryOut.DSGnrCalledArmPnpParameter.DSA1UpPickMovement.lrZone4StartPos := ARDSStationZonePosOut[iBufferPickStationNo].lrZone4StartPos - ARiVertArmPosOffset[DSA1fbPnpSequenceMemoryCall.Call_DsPnpSequenceMemory.ARiCallArmNo[iProductRecipeStepCall]];

			DSfbGnrProductRecipeMemoryOut.DSGnrCalledArmPnpParameter.DSA1UpPickMovement.lrZone1EndPos := ARDSStationZonePosOut[iBufferPickStationNo].lrZone1EndPos - ARiVertArmPosOffset[DSA1fbPnpSequenceMemoryCall.Call_DsPnpSequenceMemory.ARiCallArmNo[iProductRecipeStepCall]];
			DSfbGnrProductRecipeMemoryOut.DSGnrCalledArmPnpParameter.DSA1UpPickMovement.lrZone2EndPos := ARDSStationZonePosOut[iBufferPickStationNo].lrZone2EndPos - ARiVertArmPosOffset[DSA1fbPnpSequenceMemoryCall.Call_DsPnpSequenceMemory.ARiCallArmNo[iProductRecipeStepCall]];
			DSfbGnrProductRecipeMemoryOut.DSGnrCalledArmPnpParameter.DSA1UpPickMovement.lrZone3EndPos := ARDSStationZonePosOut[iBufferPickStationNo].lrZone3EndPos - ARiVertArmPosOffset[DSA1fbPnpSequenceMemoryCall.Call_DsPnpSequenceMemory.ARiCallArmNo[iProductRecipeStepCall]];
			DSfbGnrProductRecipeMemoryOut.DSGnrCalledArmPnpParameter.DSA1UpPickMovement.lrZone4EndPos := ARDSStationZonePosOut[iBufferPickStationNo].lrZone4EndPos - ARiVertArmPosOffset[DSA1fbPnpSequenceMemoryCall.Call_DsPnpSequenceMemory.ARiCallArmNo[iProductRecipeStepCall]];

			DSfbGnrProductRecipeMemoryOut.DSGnrCalledArmPnpParameter.DSA1DownPickMovement.lrMidPos := ARDSStationZonePosOut[iBufferPickStationNo].lrMidPos;
			DSfbGnrProductRecipeMemoryOut.DSGnrCalledArmPnpParameter.DSA1UpPickMovement.lrMidPos := ARDSStationZonePosOut[iBufferPickStationNo].lrMidPos;

		END_IF

DSfbGnrProductRecipeMemoryOut.iCallCaseNo:=62;


END_IF


IF iBufferPickStationNo < 1 OR (NOT bPickLdStnFound AND NOT bPickUldStnFound AND  iBufferPickStationNo > iStnQty) THEN

DSfbGnrProductRecipeMemoryOut.iCallCaseNo:=83;
END_IF


(*[][][][][][][][][][][][][][][][][][][][][][][][][][][][][][][][][][][][][][][][][][][][][][][][][][][][][][][][][][][][][][][][][][][][][][][][][][][][][][][][][][][][][][][][][][][][][][][][][][][]*)






(*[][][][][][][][][][][][][][][][][][][][][][][][][][][][][][][][][][][][][][][][][][][][][][][][][][][][][][][][][][][][][][][][][][][][][][][][][][][][][][][][][][][][][][][][][][][][][][][][][][][]*)
54: (* Push UpTransfer Zone4  Velo/Acc/Dcc to UpTransfer Movement*)

DSA31ArmSpeedProfileCall.Call_iArmSpdProfile := DSBufferUpTransferPattern.iZone4SpdProfileNo;
DSA31ArmSpeedProfileCall.bCallPB := TRUE;


IF DSA31ArmSpeedProfileCall.bCallCompleted THEN
DSA31ArmSpeedProfileCall.bCallPB := FALSE;
DSfbGnrProductRecipeMemoryOut.DSGnrCalledArmPnpParameter.DSA1UpTransferMovement.lrZone4SpeedVelo := DSA31ArmSpeedProfileCall.Call_DSArmSpdProfile.lrSpeedVelo;
DSfbGnrProductRecipeMemoryOut.DSGnrCalledArmPnpParameter.DSA1UpTransferMovement.lrZone4Acc := DSA31ArmSpeedProfileCall.Call_DSArmSpdProfile.lrAcc;
DSfbGnrProductRecipeMemoryOut.DSGnrCalledArmPnpParameter.DSA1UpTransferMovement.lrZone4Dcc := DSA31ArmSpeedProfileCall.Call_DSArmSpdProfile.lrDcc;

DSfbGnrProductRecipeMemoryOut.iCallCaseNo:=61;
END_IF

IF rebInvalidSpeedProfileMemoryCall.Q THEN
DSA31ArmSpeedProfileCall.bCallPB := FALSE;

DSfbGnrProductRecipeMemoryOut.iCallCaseNo:=82;
END_IF



53: (* Push UpTransfer Zone3  Velo/Acc/Dcc to UpTransfer Movement*)

DSA31ArmSpeedProfileCall.Call_iArmSpdProfile := DSBufferUpTransferPattern.iZone3SpdProfileNo;
DSA31ArmSpeedProfileCall.bCallPB := TRUE;


IF DSA31ArmSpeedProfileCall.bCallCompleted THEN
DSA31ArmSpeedProfileCall.bCallPB := FALSE;
DSfbGnrProductRecipeMemoryOut.DSGnrCalledArmPnpParameter.DSA1UpTransferMovement.lrZone3SpeedVelo := DSA31ArmSpeedProfileCall.Call_DSArmSpdProfile.lrSpeedVelo;
DSfbGnrProductRecipeMemoryOut.DSGnrCalledArmPnpParameter.DSA1UpTransferMovement.lrZone3Acc := DSA31ArmSpeedProfileCall.Call_DSArmSpdProfile.lrAcc;
DSfbGnrProductRecipeMemoryOut.DSGnrCalledArmPnpParameter.DSA1UpTransferMovement.lrZone3Dcc := DSA31ArmSpeedProfileCall.Call_DSArmSpdProfile.lrDcc;

DSfbGnrProductRecipeMemoryOut.iCallCaseNo:=54;
END_IF

IF rebInvalidSpeedProfileMemoryCall.Q THEN
DSA31ArmSpeedProfileCall.bCallPB := FALSE;

DSfbGnrProductRecipeMemoryOut.iCallCaseNo:=82;
END_IF



52: (* Push UpTransfer Zone2  Velo/Acc/Dcc to UpTransfer Movement*)

DSA31ArmSpeedProfileCall.Call_iArmSpdProfile := DSBufferUpTransferPattern.iZone2SpdProfileNo;
DSA31ArmSpeedProfileCall.bCallPB := TRUE;


IF DSA31ArmSpeedProfileCall.bCallCompleted THEN
DSA31ArmSpeedProfileCall.bCallPB := FALSE;
DSfbGnrProductRecipeMemoryOut.DSGnrCalledArmPnpParameter.DSA1UpTransferMovement.lrZone2SpeedVelo := DSA31ArmSpeedProfileCall.Call_DSArmSpdProfile.lrSpeedVelo;
DSfbGnrProductRecipeMemoryOut.DSGnrCalledArmPnpParameter.DSA1UpTransferMovement.lrZone2Acc := DSA31ArmSpeedProfileCall.Call_DSArmSpdProfile.lrAcc;
DSfbGnrProductRecipeMemoryOut.DSGnrCalledArmPnpParameter.DSA1UpTransferMovement.lrZone2Dcc := DSA31ArmSpeedProfileCall.Call_DSArmSpdProfile.lrDcc;

DSfbGnrProductRecipeMemoryOut.iCallCaseNo:=53;
END_IF

IF rebInvalidSpeedProfileMemoryCall.Q THEN
DSA31ArmSpeedProfileCall.bCallPB := FALSE;

DSfbGnrProductRecipeMemoryOut.iCallCaseNo:=82;
END_IF


51: (* Push UpTransfer Zone1  Velo/Acc/Dcc to UpTransfer Movement*)

DSA31ArmSpeedProfileCall.Call_iArmSpdProfile := DSBufferUpTransferPattern.iZone1SpdProfileNo;
DSA31ArmSpeedProfileCall.bCallPB := TRUE;


IF DSA31ArmSpeedProfileCall.bCallCompleted THEN
DSA31ArmSpeedProfileCall.bCallPB := FALSE;
DSfbGnrProductRecipeMemoryOut.DSGnrCalledArmPnpParameter.DSA1UpTransferMovement.lrZone1SpeedVelo := DSA31ArmSpeedProfileCall.Call_DSArmSpdProfile.lrSpeedVelo;
DSfbGnrProductRecipeMemoryOut.DSGnrCalledArmPnpParameter.DSA1UpTransferMovement.lrZone1Acc := DSA31ArmSpeedProfileCall.Call_DSArmSpdProfile.lrAcc;
DSfbGnrProductRecipeMemoryOut.DSGnrCalledArmPnpParameter.DSA1UpTransferMovement.lrZone1Dcc := DSA31ArmSpeedProfileCall.Call_DSArmSpdProfile.lrDcc;

DSfbGnrProductRecipeMemoryOut.iCallCaseNo:=52;
END_IF

IF rebInvalidSpeedProfileMemoryCall.Q THEN
DSA31ArmSpeedProfileCall.bCallPB := FALSE;

DSfbGnrProductRecipeMemoryOut.iCallCaseNo:=82;
END_IF

(*[][][][][][][][][][][][][][][][][][][][][][][][][][][][][][][][][][][][][][][][][][][][][][][][][][][][][][][][][][][][][][][][][][][][][][][][][][][][][][][][][][][][][][][][][][][][][][][][][][][]*)


(*[][][][][][][][][][][][][][][][][][][][][][][][][][][][][][][][][][][][][][][][][][][][][][][][][][][][][][][][][][][][][][][][][][][][][][][][][][][][][][][][][][][][][][][][][][][][][][][][][][][]*)
44: (* Push DownTransfer Zone4  Velo/Acc/Dcc to DownTransfer Movement*)

DSA31ArmSpeedProfileCall.Call_iArmSpdProfile := DSBufferDownTransferPattern.iZone4SpdProfileNo;
DSA31ArmSpeedProfileCall.bCallPB := TRUE;


IF DSA31ArmSpeedProfileCall.bCallCompleted THEN
DSA31ArmSpeedProfileCall.bCallPB := FALSE;
DSfbGnrProductRecipeMemoryOut.DSGnrCalledArmPnpParameter.DSA1DownTransferMovement.lrZone4SpeedVelo := DSA31ArmSpeedProfileCall.Call_DSArmSpdProfile.lrSpeedVelo;
DSfbGnrProductRecipeMemoryOut.DSGnrCalledArmPnpParameter.DSA1DownTransferMovement.lrZone4Acc := DSA31ArmSpeedProfileCall.Call_DSArmSpdProfile.lrAcc;
DSfbGnrProductRecipeMemoryOut.DSGnrCalledArmPnpParameter.DSA1DownTransferMovement.lrZone4Dcc := DSA31ArmSpeedProfileCall.Call_DSArmSpdProfile.lrDcc;

DSfbGnrProductRecipeMemoryOut.iCallCaseNo:=51;
END_IF

IF rebInvalidSpeedProfileMemoryCall.Q THEN
DSA31ArmSpeedProfileCall.bCallPB := FALSE;

DSfbGnrProductRecipeMemoryOut.iCallCaseNo:=82;
END_IF



43: (* Push DownTransfer Zone3  Velo/Acc/Dcc to DownTransfer Movement*)

DSA31ArmSpeedProfileCall.Call_iArmSpdProfile := DSBufferDownTransferPattern.iZone3SpdProfileNo;
DSA31ArmSpeedProfileCall.bCallPB := TRUE;


IF DSA31ArmSpeedProfileCall.bCallCompleted THEN
DSA31ArmSpeedProfileCall.bCallPB := FALSE;
DSfbGnrProductRecipeMemoryOut.DSGnrCalledArmPnpParameter.DSA1DownTransferMovement.lrZone3SpeedVelo := DSA31ArmSpeedProfileCall.Call_DSArmSpdProfile.lrSpeedVelo;
DSfbGnrProductRecipeMemoryOut.DSGnrCalledArmPnpParameter.DSA1DownTransferMovement.lrZone3Acc := DSA31ArmSpeedProfileCall.Call_DSArmSpdProfile.lrAcc;
DSfbGnrProductRecipeMemoryOut.DSGnrCalledArmPnpParameter.DSA1DownTransferMovement.lrZone3Dcc := DSA31ArmSpeedProfileCall.Call_DSArmSpdProfile.lrDcc;

DSfbGnrProductRecipeMemoryOut.iCallCaseNo:=44;
END_IF

IF rebInvalidSpeedProfileMemoryCall.Q THEN
DSA31ArmSpeedProfileCall.bCallPB := FALSE;

DSfbGnrProductRecipeMemoryOut.iCallCaseNo:=82;
END_IF



42: (* Push DownTransfer Zone2  Velo/Acc/Dcc to DownTransfer Movement*)

DSA31ArmSpeedProfileCall.Call_iArmSpdProfile := DSBufferDownTransferPattern.iZone2SpdProfileNo;
DSA31ArmSpeedProfileCall.bCallPB := TRUE;


IF DSA31ArmSpeedProfileCall.bCallCompleted THEN
DSA31ArmSpeedProfileCall.bCallPB := FALSE;
DSfbGnrProductRecipeMemoryOut.DSGnrCalledArmPnpParameter.DSA1DownTransferMovement.lrZone2SpeedVelo := DSA31ArmSpeedProfileCall.Call_DSArmSpdProfile.lrSpeedVelo;
DSfbGnrProductRecipeMemoryOut.DSGnrCalledArmPnpParameter.DSA1DownTransferMovement.lrZone2Acc := DSA31ArmSpeedProfileCall.Call_DSArmSpdProfile.lrAcc;
DSfbGnrProductRecipeMemoryOut.DSGnrCalledArmPnpParameter.DSA1DownTransferMovement.lrZone2Dcc := DSA31ArmSpeedProfileCall.Call_DSArmSpdProfile.lrDcc;

DSfbGnrProductRecipeMemoryOut.iCallCaseNo:=43;
END_IF

IF rebInvalidSpeedProfileMemoryCall.Q THEN
DSA31ArmSpeedProfileCall.bCallPB := FALSE;

DSfbGnrProductRecipeMemoryOut.iCallCaseNo:=82;
END_IF


41: (* Push DownTransfer Zone1  Velo/Acc/Dcc to DownTransfer Movement*)

DSA31ArmSpeedProfileCall.Call_iArmSpdProfile := DSBufferDownTransferPattern.iZone1SpdProfileNo;
DSA31ArmSpeedProfileCall.bCallPB := TRUE;


IF DSA31ArmSpeedProfileCall.bCallCompleted THEN
DSA31ArmSpeedProfileCall.bCallPB := FALSE;
DSfbGnrProductRecipeMemoryOut.DSGnrCalledArmPnpParameter.DSA1DownTransferMovement.lrZone1SpeedVelo := DSA31ArmSpeedProfileCall.Call_DSArmSpdProfile.lrSpeedVelo;
DSfbGnrProductRecipeMemoryOut.DSGnrCalledArmPnpParameter.DSA1DownTransferMovement.lrZone1Acc := DSA31ArmSpeedProfileCall.Call_DSArmSpdProfile.lrAcc;
DSfbGnrProductRecipeMemoryOut.DSGnrCalledArmPnpParameter.DSA1DownTransferMovement.lrZone1Dcc := DSA31ArmSpeedProfileCall.Call_DSArmSpdProfile.lrDcc;

DSfbGnrProductRecipeMemoryOut.iCallCaseNo:=42;
END_IF

IF rebInvalidSpeedProfileMemoryCall.Q THEN
DSA31ArmSpeedProfileCall.bCallPB := FALSE;

DSfbGnrProductRecipeMemoryOut.iCallCaseNo:=82;
END_IF

(*[][][][][][][][][][][][][][][][][][][][][][][][][][][][][][][][][][][][][][][][][][][][][][][][][][][][][][][][][][][][][][][][][][][][][][][][][][][][][][][][][][][][][][][][][][][][][][][][][][][]*)

(*[][][][][][][][][][][][][][][][][][][][][][][][][][][][][][][][][][][][][][][][][][][][][][][][][][][][][][][][][][][][][][][][][][][][][][][][][][][][][][][][][][][][][][][][][][][][][][][][][][][]*)
34: (* Push UpPick Zone4  Velo/Acc/Dcc to UpPick Movement*)

DSA31ArmSpeedProfileCall.Call_iArmSpdProfile := DSBufferUpPickPattern.iZone4SpdProfileNo;
DSA31ArmSpeedProfileCall.bCallPB := TRUE;


IF DSA31ArmSpeedProfileCall.bCallCompleted THEN
DSA31ArmSpeedProfileCall.bCallPB := FALSE;
DSfbGnrProductRecipeMemoryOut.DSGnrCalledArmPnpParameter.DSA1UpPickMovement.lrZone4SpeedVelo := DSA31ArmSpeedProfileCall.Call_DSArmSpdProfile.lrSpeedVelo;
DSfbGnrProductRecipeMemoryOut.DSGnrCalledArmPnpParameter.DSA1UpPickMovement.lrZone4Acc := DSA31ArmSpeedProfileCall.Call_DSArmSpdProfile.lrAcc;
DSfbGnrProductRecipeMemoryOut.DSGnrCalledArmPnpParameter.DSA1UpPickMovement.lrZone4Dcc := DSA31ArmSpeedProfileCall.Call_DSArmSpdProfile.lrDcc;

DSfbGnrProductRecipeMemoryOut.iCallCaseNo:=41;
END_IF

IF rebInvalidSpeedProfileMemoryCall.Q THEN
DSA31ArmSpeedProfileCall.bCallPB := FALSE;

DSfbGnrProductRecipeMemoryOut.iCallCaseNo:=82;
END_IF



33: (* Push UpPick Zone3  Velo/Acc/Dcc to UpPick Movement*)

DSA31ArmSpeedProfileCall.Call_iArmSpdProfile := DSBufferUpPickPattern.iZone3SpdProfileNo;
DSA31ArmSpeedProfileCall.bCallPB := TRUE;


IF DSA31ArmSpeedProfileCall.bCallCompleted THEN
DSA31ArmSpeedProfileCall.bCallPB := FALSE;
DSfbGnrProductRecipeMemoryOut.DSGnrCalledArmPnpParameter.DSA1UpPickMovement.lrZone3SpeedVelo := DSA31ArmSpeedProfileCall.Call_DSArmSpdProfile.lrSpeedVelo;
DSfbGnrProductRecipeMemoryOut.DSGnrCalledArmPnpParameter.DSA1UpPickMovement.lrZone3Acc := DSA31ArmSpeedProfileCall.Call_DSArmSpdProfile.lrAcc;
DSfbGnrProductRecipeMemoryOut.DSGnrCalledArmPnpParameter.DSA1UpPickMovement.lrZone3Dcc := DSA31ArmSpeedProfileCall.Call_DSArmSpdProfile.lrDcc;

DSfbGnrProductRecipeMemoryOut.iCallCaseNo:=34;
END_IF

IF rebInvalidSpeedProfileMemoryCall.Q THEN
DSA31ArmSpeedProfileCall.bCallPB := FALSE;

DSfbGnrProductRecipeMemoryOut.iCallCaseNo:=82;
END_IF



32: (* Push UpPick Zone2  Velo/Acc/Dcc to UpPick Movement*)

DSA31ArmSpeedProfileCall.Call_iArmSpdProfile := DSBufferUpPickPattern.iZone2SpdProfileNo;
DSA31ArmSpeedProfileCall.bCallPB := TRUE;


IF DSA31ArmSpeedProfileCall.bCallCompleted THEN
DSA31ArmSpeedProfileCall.bCallPB := FALSE;
DSfbGnrProductRecipeMemoryOut.DSGnrCalledArmPnpParameter.DSA1UpPickMovement.lrZone2SpeedVelo := DSA31ArmSpeedProfileCall.Call_DSArmSpdProfile.lrSpeedVelo;
DSfbGnrProductRecipeMemoryOut.DSGnrCalledArmPnpParameter.DSA1UpPickMovement.lrZone2Acc := DSA31ArmSpeedProfileCall.Call_DSArmSpdProfile.lrAcc;
DSfbGnrProductRecipeMemoryOut.DSGnrCalledArmPnpParameter.DSA1UpPickMovement.lrZone2Dcc := DSA31ArmSpeedProfileCall.Call_DSArmSpdProfile.lrDcc;

DSfbGnrProductRecipeMemoryOut.iCallCaseNo:=33;
END_IF

IF rebInvalidSpeedProfileMemoryCall.Q THEN
DSA31ArmSpeedProfileCall.bCallPB := FALSE;

DSfbGnrProductRecipeMemoryOut.iCallCaseNo:=82;
END_IF


31: (* Push UpPick Zone1  Velo/Acc/Dcc to UpPick Movement*)

DSA31ArmSpeedProfileCall.Call_iArmSpdProfile := DSBufferUpPickPattern.iZone1SpdProfileNo;
DSA31ArmSpeedProfileCall.bCallPB := TRUE;


IF DSA31ArmSpeedProfileCall.bCallCompleted THEN
DSA31ArmSpeedProfileCall.bCallPB := FALSE;
DSfbGnrProductRecipeMemoryOut.DSGnrCalledArmPnpParameter.DSA1UpPickMovement.lrZone1SpeedVelo := DSA31ArmSpeedProfileCall.Call_DSArmSpdProfile.lrSpeedVelo;
DSfbGnrProductRecipeMemoryOut.DSGnrCalledArmPnpParameter.DSA1UpPickMovement.lrZone1Acc := DSA31ArmSpeedProfileCall.Call_DSArmSpdProfile.lrAcc;
DSfbGnrProductRecipeMemoryOut.DSGnrCalledArmPnpParameter.DSA1UpPickMovement.lrZone1Dcc := DSA31ArmSpeedProfileCall.Call_DSArmSpdProfile.lrDcc;

DSfbGnrProductRecipeMemoryOut.iCallCaseNo:=32;
END_IF

IF rebInvalidSpeedProfileMemoryCall.Q THEN
DSA31ArmSpeedProfileCall.bCallPB := FALSE;

DSfbGnrProductRecipeMemoryOut.iCallCaseNo:=82;
END_IF

(*[][][][][][][][][][][][][][][][][][][][][][][][][][][][][][][][][][][][][][][][][][][][][][][][][][][][][][][][][][][][][][][][][][][][][][][][][][][][][][][][][][][][][][][][][][][][][][][][][][][]*)


(*[][][][][][][][][][][][][][][][][][][][][][][][][][][][][][][][][][][][][][][][][][][][][][][][][][][][][][][][][][][][][][][][][][][][][][][][][][][][][][][][][][][][][][][][][][][][][][][][][][][]*)
24: (* Push DownPick Zone4  Velo/Acc/Dcc to DownPick Movement*)

DSA31ArmSpeedProfileCall.Call_iArmSpdProfile := DSBufferDownPickPattern.iZone4SpdProfileNo;
DSA31ArmSpeedProfileCall.bCallPB := TRUE;


IF DSA31ArmSpeedProfileCall.bCallCompleted THEN
DSA31ArmSpeedProfileCall.bCallPB := FALSE;
DSfbGnrProductRecipeMemoryOut.DSGnrCalledArmPnpParameter.DSA1DownPickMovement.lrZone4SpeedVelo := DSA31ArmSpeedProfileCall.Call_DSArmSpdProfile.lrSpeedVelo;
DSfbGnrProductRecipeMemoryOut.DSGnrCalledArmPnpParameter.DSA1DownPickMovement.lrZone4Acc := DSA31ArmSpeedProfileCall.Call_DSArmSpdProfile.lrAcc;
DSfbGnrProductRecipeMemoryOut.DSGnrCalledArmPnpParameter.DSA1DownPickMovement.lrZone4Dcc := DSA31ArmSpeedProfileCall.Call_DSArmSpdProfile.lrDcc;

DSfbGnrProductRecipeMemoryOut.iCallCaseNo:=31;
END_IF

IF rebInvalidSpeedProfileMemoryCall.Q THEN
DSA31ArmSpeedProfileCall.bCallPB := FALSE;

DSfbGnrProductRecipeMemoryOut.iCallCaseNo:=82;
END_IF



23: (* Push DownPick Zone3  Velo/Acc/Dcc to DownPick Movement*)

DSA31ArmSpeedProfileCall.Call_iArmSpdProfile := DSBufferDownPickPattern.iZone3SpdProfileNo;
DSA31ArmSpeedProfileCall.bCallPB := TRUE;


IF DSA31ArmSpeedProfileCall.bCallCompleted THEN
DSA31ArmSpeedProfileCall.bCallPB := FALSE;
DSfbGnrProductRecipeMemoryOut.DSGnrCalledArmPnpParameter.DSA1DownPickMovement.lrZone3SpeedVelo := DSA31ArmSpeedProfileCall.Call_DSArmSpdProfile.lrSpeedVelo;
DSfbGnrProductRecipeMemoryOut.DSGnrCalledArmPnpParameter.DSA1DownPickMovement.lrZone3Acc := DSA31ArmSpeedProfileCall.Call_DSArmSpdProfile.lrAcc;
DSfbGnrProductRecipeMemoryOut.DSGnrCalledArmPnpParameter.DSA1DownPickMovement.lrZone3Dcc := DSA31ArmSpeedProfileCall.Call_DSArmSpdProfile.lrDcc;

DSfbGnrProductRecipeMemoryOut.iCallCaseNo:=24;
END_IF

IF rebInvalidSpeedProfileMemoryCall.Q THEN
DSA31ArmSpeedProfileCall.bCallPB := FALSE;

DSfbGnrProductRecipeMemoryOut.iCallCaseNo:=82;
END_IF



22: (* Push DownPick Zone2  Velo/Acc/Dcc to DownPick Movement*)

DSA31ArmSpeedProfileCall.Call_iArmSpdProfile := DSBufferDownPickPattern.iZone2SpdProfileNo;
DSA31ArmSpeedProfileCall.bCallPB := TRUE;


IF DSA31ArmSpeedProfileCall.bCallCompleted THEN
DSA31ArmSpeedProfileCall.bCallPB := FALSE;
DSfbGnrProductRecipeMemoryOut.DSGnrCalledArmPnpParameter.DSA1DownPickMovement.lrZone2SpeedVelo := DSA31ArmSpeedProfileCall.Call_DSArmSpdProfile.lrSpeedVelo;
DSfbGnrProductRecipeMemoryOut.DSGnrCalledArmPnpParameter.DSA1DownPickMovement.lrZone2Acc := DSA31ArmSpeedProfileCall.Call_DSArmSpdProfile.lrAcc;
DSfbGnrProductRecipeMemoryOut.DSGnrCalledArmPnpParameter.DSA1DownPickMovement.lrZone2Dcc := DSA31ArmSpeedProfileCall.Call_DSArmSpdProfile.lrDcc;

DSfbGnrProductRecipeMemoryOut.iCallCaseNo:=23;
END_IF

IF rebInvalidSpeedProfileMemoryCall.Q THEN
DSA31ArmSpeedProfileCall.bCallPB := FALSE;

DSfbGnrProductRecipeMemoryOut.iCallCaseNo:=82;
END_IF


21: (* Push DownPick Zone1  Velo/Acc/Dcc to DownPick Movement*)

DSA31ArmSpeedProfileCall.Call_iArmSpdProfile := DSBufferDownPickPattern.iZone1SpdProfileNo;
DSA31ArmSpeedProfileCall.bCallPB := TRUE;


IF DSA31ArmSpeedProfileCall.bCallCompleted THEN
DSA31ArmSpeedProfileCall.bCallPB := FALSE;
DSfbGnrProductRecipeMemoryOut.DSGnrCalledArmPnpParameter.DSA1DownPickMovement.lrZone1SpeedVelo := DSA31ArmSpeedProfileCall.Call_DSArmSpdProfile.lrSpeedVelo;
DSfbGnrProductRecipeMemoryOut.DSGnrCalledArmPnpParameter.DSA1DownPickMovement.lrZone1Acc := DSA31ArmSpeedProfileCall.Call_DSArmSpdProfile.lrAcc;
DSfbGnrProductRecipeMemoryOut.DSGnrCalledArmPnpParameter.DSA1DownPickMovement.lrZone1Dcc := DSA31ArmSpeedProfileCall.Call_DSArmSpdProfile.lrDcc;

DSfbGnrProductRecipeMemoryOut.iCallCaseNo:=22;
END_IF

IF rebInvalidSpeedProfileMemoryCall.Q THEN
DSA31ArmSpeedProfileCall.bCallPB := FALSE;

DSfbGnrProductRecipeMemoryOut.iCallCaseNo:=82;
END_IF

(*[][][][][][][][][][][][][][][][][][][][][][][][][][][][][][][][][][][][][][][][][][][][][][][][][][][][][][][][][][][][][][][][][][][][][][][][][][][][][][][][][][][][][][][][][][][][][][][][][][][]*)



14: (* Call UpPickPattern*)
DSA21UpDownPatternCall.Call_iUpDownPatternNo := DSA1fbPnpSequenceMemoryCall.Call_DsPnpSequenceMemory.ARiUpTransferPatternNo[iProductRecipeStepCall];
DSA21UpDownPatternCall.bCallPB := TRUE;


IF DSA21UpDownPatternCall.bCallCompleted THEN
DSA21UpDownPatternCall.bCallPB := FALSE;
DSBufferUpTransferPattern := DSA21UpDownPatternCall.Call_DsUpDownPattern;
DSfbGnrProductRecipeMemoryOut.DSGnrCalledArmPnpParameter.DSA1UpTransferMovement.sUpDownPatternDescription := DSA21UpDownPatternCall.Call_DsUpDownPattern.sDescription;
DSfbGnrProductRecipeMemoryOut.iCallCaseNo:=21;
END_IF

13: (* Call DownTransferPattern*)
DSA21UpDownPatternCall.Call_iUpDownPatternNo := DSA1fbPnpSequenceMemoryCall.Call_DsPnpSequenceMemory.ARiDownTransferPatternNo[iProductRecipeStepCall];
DSA21UpDownPatternCall.bCallPB := TRUE;


IF DSA21UpDownPatternCall.bCallCompleted THEN
DSA21UpDownPatternCall.bCallPB := FALSE;
DSBufferDownTransferPattern := DSA21UpDownPatternCall.Call_DsUpDownPattern;
DSfbGnrProductRecipeMemoryOut.DSGnrCalledArmPnpParameter.DSA1DownTransferMovement.sUpDownPatternDescription := DSA21UpDownPatternCall.Call_DsUpDownPattern.sDescription;
DSfbGnrProductRecipeMemoryOut.iCallCaseNo:=14;
END_IF

IF rebInvalidUpDownPatternMemoryCall.Q THEN
DSA21UpDownPatternCall.bCallPB := FALSE;

DSfbGnrProductRecipeMemoryOut.iCallCaseNo:=81;
END_IF

12: (* Call UpPickPattern*)
DSA21UpDownPatternCall.Call_iUpDownPatternNo := DSA1fbPnpSequenceMemoryCall.Call_DsPnpSequenceMemory.ARiUpPickPatternNo[iProductRecipeStepCall];
DSA21UpDownPatternCall.bCallPB := TRUE;


IF DSA21UpDownPatternCall.bCallCompleted THEN
DSA21UpDownPatternCall.bCallPB := FALSE;
DSBufferUpPickPattern := DSA21UpDownPatternCall.Call_DsUpDownPattern;
DSfbGnrProductRecipeMemoryOut.DSGnrCalledArmPnpParameter.DSA1UpPickMovement.sUpDownPatternDescription := DSA21UpDownPatternCall.Call_DsUpDownPattern.sDescription;
DSfbGnrProductRecipeMemoryOut.iCallCaseNo:=13;
END_IF

IF rebInvalidUpDownPatternMemoryCall.Q THEN
DSA21UpDownPatternCall.bCallPB := FALSE;

DSfbGnrProductRecipeMemoryOut.iCallCaseNo:=81;
END_IF

11: (* Call DownPickPattern*)
DSA21UpDownPatternCall.Call_iUpDownPatternNo := DSA1fbPnpSequenceMemoryCall.Call_DsPnpSequenceMemory.ARiDownPickPatternNo[iProductRecipeStepCall];
DSA21UpDownPatternCall.bCallPB := TRUE;


IF DSA21UpDownPatternCall.bCallCompleted THEN
DSA21UpDownPatternCall.bCallPB := FALSE;
DSBufferDownPickPattern := DSA21UpDownPatternCall.Call_DsUpDownPattern;
DSfbGnrProductRecipeMemoryOut.DSGnrCalledArmPnpParameter.DSA1DownPickMovement.sUpDownPatternDescription := DSA21UpDownPatternCall.Call_DsUpDownPattern.sDescription;
DSfbGnrProductRecipeMemoryOut.iCallCaseNo:=12;
END_IF

IF rebInvalidUpDownPatternMemoryCall.Q THEN
DSA21UpDownPatternCall.bCallPB := FALSE;

DSfbGnrProductRecipeMemoryOut.iCallCaseNo:=81;
END_IF


10: (*Push UpDownPattern to Buffer*)
iBufferPickStationNo := DSA1fbPnpSequenceMemoryCall.Call_DsPnpSequenceMemory.ARiPickStationNo[iProductRecipeStepCall];
iBufferTransferStationNo := DSA1fbPnpSequenceMemoryCall.Call_DsPnpSequenceMemory.ARiTransferStationNo[iProductRecipeStepCall];

iBufferDownPickPatternNo := DSA1fbPnpSequenceMemoryCall.Call_DsPnpSequenceMemory.ARiDownPickPatternNo[iProductRecipeStepCall];
iBufferUpPickPatternNo := DSA1fbPnpSequenceMemoryCall.Call_DsPnpSequenceMemory.ARiUpPickPatternNo[iProductRecipeStepCall];
iBufferDownTransferPatternNo := DSA1fbPnpSequenceMemoryCall.Call_DsPnpSequenceMemory.ARiDownTransferPatternNo[iProductRecipeStepCall];
iBufferUpTransferPatternNo := DSA1fbPnpSequenceMemoryCall.Call_DsPnpSequenceMemory.ARiUpTransferPatternNo[iProductRecipeStepCall];

DSfbGnrProductRecipeMemoryOut.DSGnrCalledArmPnpParameter.iStnSeqRecipeNo := DSA1fbPnpSequenceMemoryCall.Call_DsPnpSequenceMemory.ARiStnSeqRepNo[iProductRecipeStepCall];
DSfbGnrProductRecipeMemoryOut.DSGnrCalledArmPnpParameter.iLdGroupNo := DSA1fbPnpSequenceMemoryCall.Call_DsPnpSequenceMemory.iLdGroupNo;
DSfbGnrProductRecipeMemoryOut.DSGnrCalledArmPnpParameter.iUldGroupNo := DSA1fbPnpSequenceMemoryCall.Call_DsPnpSequenceMemory.iUldGroupNo;


DSfbGnrProductRecipeMemoryOut.sProductRecipeDescription := DSA1fbPnpSequenceMemoryCall.Call_DsPnpSequenceMemory.sDescription;

DSfbGnrProductRecipeMemoryOut.iCallCaseNo:=11;


71: (*Complete Data Called*)

	IF bEnableCallArmNo THEN
	DSfbGnrProductRecipeMemoryOut.DSGnrCalledArmPnpParameter.iCallArmNo := iCallArmNo;
	ELSE
	DSfbGnrProductRecipeMemoryOut.DSGnrCalledArmPnpParameter.iCallArmNo := DSA1fbPnpSequenceMemoryCall.Call_DsPnpSequenceMemory.ARiCallArmNo[iProductRecipeStepCall];
	END_IF

DSfbGnrProductRecipeMemoryOut.bCallCompleted := TRUE;
CallSelfCheckHR := FALSE;
DSfbGnrProductRecipeMemoryOut.iCallCaseNo:=72;

72:; (*Done without error*)

81:
(*iPreviousProcessStep := iCurrentProcessStep;*)
CallSelfCheckHR := FALSE;
DSfbGnrProductRecipeMemoryOut.bCallUpDownPatternMemoryErr := TRUE;
DSfbGnrProductRecipeMemoryOut.iCallCaseNo:=91;

82:
(*iPreviousProcessStep := iCurrentProcessStep;*)
DSfbGnrProductRecipeMemoryOut.bCallArmSpeedProfileMemoryErr := TRUE;
CallSelfCheckHR := FALSE;
DSfbGnrProductRecipeMemoryOut.iCallCaseNo:=92;

83:
(*iPreviousProcessStep := iCurrentProcessStep;*)
DSfbGnrProductRecipeMemoryOut.bCallPickStationNoErr := TRUE;
CallSelfCheckHR := FALSE;
DSfbGnrProductRecipeMemoryOut.iCallCaseNo:=93;

84:
(*iPreviousProcessStep := iCurrentProcessStep;*)
DSfbGnrProductRecipeMemoryOut.bCallTransferStationNoErr := TRUE;
CallSelfCheckHR := FALSE;
DSfbGnrProductRecipeMemoryOut.iCallCaseNo:=94;



91:; (*Found UpDownPatternMemoryError and Task Not Complete *)

92:; (*Found ArmSpeedProfileMemoryErr and Task Not Complete *)

93:; (*Found PickStationNoErr and Task Not Complete *)

94:; (*Found TransferStationNoErr and Task Not Complete *)



END_CASE

END_FUNCTION_BLOCK

// ---- FBs/B_JKS_NewFB_V2/FBP-Memory_Sub/fbV2_A1_PnpSequenceMemory.TcPOU
FUNCTION_BLOCK fbV2_A1_PnpSequenceMemory

VAR CONSTANT
END_VAR

VAR_INPUT
	bSavePB  : BOOL;
	bLoadPB  : BOOL;
	bClearPB : BOOL;
	bCopyPB  : BOOL;
	iCopyToProductRecipeNo : INT;
(*	ARiLdStnID: INT;
	ARiUldStnID: INT;
*)END_VAR


VAR_IN_OUT PERSISTENT

	iProductRecipeNo: INT; (* 10 sets of UpDownPattern *)
	DSA1inPnpSequenceMemory : DSV2_A1_PnpSequenceMemory;

	Call_iProductRecipeNo : INT;
	bCallPB: BOOL;

END_VAR
VAR_OUTPUT
	bSaveInd: BOOL;
	bLoadInd: BOOL;
	bClearInd: BOOL;
	bCallCompleted : BOOL;
	bInvalidCallProductRecipeNoHold: BOOL;
	bInvalidCallProductRecipeNoPulse: BOOL;
	Call_DSA1PnpSequenceMemory : DSV2_A1_PnpSequenceMemory;

END_VAR
VAR
	SaveIndHr: BOOL;
	LoadIndHr: BOOL;
	ClearIndHr: BOOL;

	SaveTimerDelay  : TON;
	LoadTimerDelay  : TON;
	ClearTimerDelay : TON;
	SelfCheckTimer  : TON;
	bLoadEn: BOOL;
	SelfCheckloopPnpSequence: BOOL;

	ClearDF  : R_TRIG;
	LoadDF   : R_TRIG;
	LoadENDF : R_TRIG;

	SaveDF: R_TRIG;
	CallIntervalTimer: TON;
	CallIntervalDIFU: R_TRIG;

	bCallCompletedHR: BOOL;
	bCallCompletedHRRE: R_TRIG;
	CallCompletedTimer: TON;
	CallSelfCheckTimer : TON;
	CallSelfCheckloop : BOOL;

	CallSelfCheckRE: R_TRIG;
	CallStep: INT;
	CallSelfCheckHR: BOOL;
	bCallPBRE: R_TRIG;

	LoadFL: INT;
	SaveFL: INT;
	CallSFL: INT;
	febInvalidCallProductRecipeNo: F_TRIG;



	rebInvalidCallProductRecipeNo: R_TRIG;
	CopyDF: R_TRIG;
	PreviousProductRecipeNo: INT;
	PreviousProductRecipeCallNo: INT;
	tInvalidCallProductRecipeNoPulseTimer: TON;
	iFixPickStnFL: INT;
	iCtrlTransferStnFL: INT;
	bTransferStnEndDetected: BOOL;
	iUldStnStepNo: INT;
	iCtrlZeroB4UldStnFL: INT;
	iMaxMinFL: INT;
	iWriteEmptyDesFL: INT;
	iFL: INT;
	
	ARDsPnpSequenceMemory_Empty : DSV2_A1_PnpSequenceMemory;
END_VAR

VAR PERSISTENT

	ARDsPnpSequenceMemory : ARRAY [1..iProductRecipeArrayQty] OF DSV2_A1_PnpSequenceMemory;
	ARsStoragePnpSequenceDescription: ARRAY [0..iProductRecipeArrayQty] OF STRING(50);
	fbV2DualArmProductRecipeStnAndArmNoCtrl_General: fbV2_DualArmProductRecipeStnAndArmNoCtrl;


END_VAR




XML_ImportExport();



IF iProductRecipeNo < 1 THEN
iProductRecipeNo := 1;
END_IF

IF iProductRecipeNo > iProductRecipeArrayQty THEN
iProductRecipeNo := iProductRecipeArrayQty;
END_IF
(*Fix Pick Station No*)
DSA1inPnpSequenceMemory.ARiPickStationNo[1] := ARiLdStnID[DSA1inPnpSequenceMemory.iLdGroupNo];
iFixPickStnFL := 1;

	FOR iFixPickStnFL := 1 TO iProductRecipeStepArrayQty DO

		IF iFixPickStnFL >=1 AND iFixPickStnFL <= iProductRecipeStepArrayQty-1THEN

			IF DSA1inPnpSequenceMemory.ARiTransferStationNo[iFixPickStnFL] <> ARiUldStnID[DSA1inPnpSequenceMemory.iUldGroupNo] THEN
			DSA1inPnpSequenceMemory.ARiPickStationNo[iFixPickStnFL+1]:= DSA1inPnpSequenceMemory.ARiTransferStationNo[iFixPickStnFL];
			END_IF

			IF DSA1inPnpSequenceMemory.ARiTransferStationNo[iFixPickStnFL] = ARiUldStnID[DSA1inPnpSequenceMemory.iUldGroupNo] THEN
			DSA1inPnpSequenceMemory.ARiPickStationNo[iFixPickStnFL+1]:= 0;
			END_IF

		END_IF

	END_FOR

(*Control Transfer Station No*)
iCtrlTransferStnFL := 1;
bTransferStnEndDetected := FALSE;
iUldStnStepNo := 0;
	FOR iCtrlTransferStnFL := 1 TO iProductRecipeStepArrayQty DO

		IF iCtrlTransferStnFL >=1 AND iCtrlTransferStnFL <= iProductRecipeStepArrayQty THEN

			IF NOT bTransferStnEndDetected AND DSA1inPnpSequenceMemory.ARiTransferStationNo[iCtrlTransferStnFL] > iStnQty THEN
			DSA1inPnpSequenceMemory.ARiTransferStationNo[iCtrlTransferStnFL]:= ARiUldStnID[DSA1inPnpSequenceMemory.iUldGroupNo];
			END_IF

			IF bTransferStnEndDetected THEN
			DSA1inPnpSequenceMemory.ARiTransferStationNo[iCtrlTransferStnFL] := ARiUldStnID[DSA1inPnpSequenceMemory.iUldGroupNo](*0*);
			END_IF

			IF DSA1inPnpSequenceMemory.ARiTransferStationNo[iCtrlTransferStnFL-1] = ARiUldStnID[DSA1inPnpSequenceMemory.iUldGroupNo] THEN
			DSA1inPnpSequenceMemory.ARiTransferStationNo[iCtrlTransferStnFL] := ARiUldStnID[DSA1inPnpSequenceMemory.iUldGroupNo](*0*);
			bTransferStnEndDetected := TRUE;
			iUldStnStepNo := iCtrlTransferStnFL-1;
			END_IF

		END_IF

	END_FOR

(*No "0" before Unloading Stn Ctrl*)

IF bTransferStnEndDetected AND iUldStnStepNo > 1 THEN
iCtrlZeroB4UldStnFL := 1;

	FOR iCtrlZeroB4UldStnFL := 1 TO iUldStnStepNo DO

		IF iCtrlZeroB4UldStnFL >=1 AND iCtrlZeroB4UldStnFL <= iUldStnStepNo-1 THEN

			IF DSA1inPnpSequenceMemory.ARiTransferStationNo[iCtrlZeroB4UldStnFL] <= 0 THEN
			DSA1inPnpSequenceMemory.ARiTransferStationNo[iCtrlZeroB4UldStnFL]:= 1;
			END_IF

		END_IF

	END_FOR

END_IF


(*Min / Max Control*)
iMaxMinFL := 1;
	FOR iMaxMinFL := 1 TO iProductRecipeStepArrayQty DO

		IF iMaxMinFL >=1 AND iMaxMinFL <= iProductRecipeStepArrayQty THEN

			IF DSA1inPnpSequenceMemory.ARiDownPickPatternNo[iMaxMinFL] <= 0 THEN
			DSA1inPnpSequenceMemory.ARiDownPickPatternNo[iMaxMinFL]:= 1;
			ELSIF DSA1inPnpSequenceMemory.ARiDownPickPatternNo[iMaxMinFL] > iArmUpDownPatternArrayQty THEN
			DSA1inPnpSequenceMemory.ARiDownPickPatternNo[iMaxMinFL]:= iArmUpDownPatternArrayQty;
			END_IF

			IF DSA1inPnpSequenceMemory.ARiUpPickPatternNo[iMaxMinFL] <= 0 THEN
			DSA1inPnpSequenceMemory.ARiUpPickPatternNo[iMaxMinFL]:= 1;
			ELSIF DSA1inPnpSequenceMemory.ARiUpPickPatternNo[iMaxMinFL] > iArmUpDownPatternArrayQty THEN
			DSA1inPnpSequenceMemory.ARiUpPickPatternNo[iMaxMinFL]:= iArmUpDownPatternArrayQty;
			END_IF

			IF DSA1inPnpSequenceMemory.ARiDownTransferPatternNo[iMaxMinFL] <= 0 THEN
			DSA1inPnpSequenceMemory.ARiDownTransferPatternNo[iMaxMinFL]:= 1;
			ELSIF DSA1inPnpSequenceMemory.ARiDownTransferPatternNo[iMaxMinFL] > iArmUpDownPatternArrayQty THEN
			DSA1inPnpSequenceMemory.ARiDownTransferPatternNo[iMaxMinFL]:= iArmUpDownPatternArrayQty;
			END_IF

			IF DSA1inPnpSequenceMemory.ARiUpTransferPatternNo[iMaxMinFL] <= 0 THEN
			DSA1inPnpSequenceMemory.ARiUpTransferPatternNo[iMaxMinFL]:= 1;
			ELSIF DSA1inPnpSequenceMemory.ARiUpTransferPatternNo[iMaxMinFL] > iArmUpDownPatternArrayQty THEN
			DSA1inPnpSequenceMemory.ARiUpTransferPatternNo[iMaxMinFL]:= iArmUpDownPatternArrayQty;
			END_IF

(*			IF DSA1inPnpSequenceMemory.ARiRepeatUpDownCycle[iMaxMinFL] <= 0 THEN
			DSA1inPnpSequenceMemory.ARiRepeatUpDownCycle[iMaxMinFL]:= 1;
			ELS*)IF DSA1inPnpSequenceMemory.ARiRepeatUpDownCycle[iMaxMinFL] > 99 THEN
			DSA1inPnpSequenceMemory.ARiRepeatUpDownCycle[iMaxMinFL]:= 99;
			END_IF

			IF DSA1inPnpSequenceMemory.ARiCallArmNo[iMaxMinFL] <= 0 THEN
			DSA1inPnpSequenceMemory.ARiCallArmNo[iMaxMinFL]:= 1;
			ELSIF DSA1inPnpSequenceMemory.ARiCallArmNo[iMaxMinFL] > iArmQty THEN
			DSA1inPnpSequenceMemory.ARiCallArmNo[iMaxMinFL]:= iArmQty;
			END_IF

			IF DSA1inPnpSequenceMemory.ARiStnSeqRepNo[iMaxMinFL] <= 0 THEN
			DSA1inPnpSequenceMemory.ARiStnSeqRepNo[iMaxMinFL]:= 1;
			ELSIF DSA1inPnpSequenceMemory.ARiStnSeqRepNo[iMaxMinFL] > iStationSequenceRecipeArrayQty THEN
			DSA1inPnpSequenceMemory.ARiStnSeqRepNo[iMaxMinFL]:= iStationSequenceRecipeArrayQty;
			END_IF

		END_IF

	END_FOR


fbV2DualArmProductRecipeStnAndArmNoCtrl_General(bEN:=TRUE , DSPnpSequenceMemory:=DSA1inPnpSequenceMemory );

(*Clear Indicator*)
IF bClearPB THEN
ClearIndHr := TRUE;
END_IF

ClearTimerDelay(IN:=ClearIndHr, PT := T#1S, Q=>, ET=>);
IF ClearTimerDelay.Q THEN
ClearIndHr := FALSE;
END_IF

IF ClearIndHr AND NOT ClearTimerDelay.Q THEN
bClearInd := TRUE;
ELSE
bClearInd := FALSE;
END_IF

(*Load and Save Indicator*)
IF bSavePB THEN
SaveIndHr := TRUE;
END_IF

SaveTimerDelay(IN:=SaveIndHr, PT := T#1s, Q=>, ET=>);
IF SaveTimerDelay.Q THEN
SaveIndHr := FALSE;
END_IF

IF SaveIndHr AND NOT SaveTimerDelay.Q THEN
bSaveInd := TRUE;
ELSE
bSaveInd := FALSE;
END_IF

IF bLoadPB THEN
LoadIndHr := TRUE;
END_IF

LoadTimerDelay(IN:=LoadIndHr, PT := T#1s, Q=>, ET=>);
IF loadtimerdelay.Q THEN
LoadIndHr := FALSE;
END_IF

IF loadIndHr AND NOT LoadTimerDelay.Q THEN
bLoadInd := TRUE;
ELSE
bLoadInd := FALSE;
END_IF

IF iProductRecipeNo <> PreviousProductRecipeNo THEN
bLoadEn := TRUE;
ELSE
bLoadEn := FALSE;
END_IF


(* Load Recipe *)

LoadDF(CLK:=bLoadPB,Q=>);
LoadENDF(CLK:=bLoadEn,Q=>);

IF LoadDF.Q OR LoadENDF.Q THEN

DSA1inPnpSequenceMemory := ARDsPnpSequenceMemory[iProductRecipeNo];
PreviousProductRecipeNo := iProductRecipeNo  ;

END_IF


(* Save Recipe *)

SaveDF(CLK:=bSavePB,Q=>);

IF SaveDF.Q THEN

ARDsPnpSequenceMemory[iProductRecipeNo] := DSA1inPnpSequenceMemory;
ARsStoragePnpSequenceDescription[iProductRecipeNo] := DSA1inPnpSequenceMemory.sDescription;

END_IF


(*Copy Recipe*)

CopyDF(CLK:=bCopyPB,Q=>);

IF CopyDF.Q THEN

ARDsPnpSequenceMemory[iCopyToProductRecipeNo] := ARDsPnpSequenceMemory[iProductRecipeNo];
ARsStoragePnpSequenceDescription[iCopyToProductRecipeNo] := ARDsPnpSequenceMemory[iProductRecipeNo].sDescription;

END_IF

(* Clear Recipe *)

ClearDF(CLK:=bClearPB,Q=>);

IF ClearDF.Q THEN

ARDsPnpSequenceMemory[iProductRecipeNo] := ARDsPnpSequenceMemory_Empty;
ARsStoragePnpSequenceDescription[iProductRecipeNo] := ARDsPnpSequenceMemory_Empty.sDescription;	

DSA1inPnpSequenceMemory:= ARDsPnpSequenceMemory_Empty;
DSA1inPnpSequenceMemory.sDescription:= ARDsPnpSequenceMemory_Empty.sDescription;
DSA1fbPnpSequenceMemoryStore.iCopyToProductRecipeNo:=0;

END_IF 

(*Write Empty for Empty description *)
ARsStoragePnpSequenceDescription[0] := ' = = = No Basket = = = ';
iWriteEmptyDesFL := 1;
FOR iWriteEmptyDesFL := 1 TO iProductRecipeArrayQty DO
	IF iWriteEmptyDesFL >= 1 AND iWriteEmptyDesFL <= iProductRecipeArrayQty THEN
		IF ARsStoragePnpSequenceDescription[iWriteEmptyDesFL] = '' THEN
		ARsStoragePnpSequenceDescription[iWriteEmptyDesFL] := ' - - -  Empty Recipe - - - ';
		END_IF
	END_IF
END_FOR




(* Call Recipe *)
(* ---- Call Recipe Complete Flag ---*)


IF NOT bCallPB THEN
bCallCompleted := FALSE;
END_IF

bCallPBRE(CLK:=bCallPB , Q=> );

IF (Call_iProductRecipeNo <= 0 OR Call_iProductRecipeNo > iProductRecipeArrayQty) AND bCallPB THEN
bInvalidCallProductRecipeNoHold := TRUE;
ELSE
bInvalidCallProductRecipeNoHold := FALSE;
END_IF


febInvalidCallProductRecipeNo(CLK:= bCallPB AND bInvalidCallProductRecipeNoHold  , Q=> );

IF febInvalidCallProductRecipeNo.Q THEN
bInvalidCallProductRecipeNoPulse := TRUE;
END_IF

tInvalidCallProductRecipeNoPulseTimer(IN:=bInvalidCallProductRecipeNoPulse , PT:=t#0.5s , Q=> , ET=> );

IF tInvalidCallProductRecipeNoPulseTimer.Q OR NOT bCallPB THEN
bInvalidCallProductRecipeNoPulse := FALSE;
END_IF

IF bCallPBRE.Q AND NOT bInvalidCallProductRecipeNoHold THEN
bCallCompleted := FALSE;
CallStep:= 1;
END_IF


CASE CallStep OF

1:

Call_DSA1PnpSequenceMemory := ARDsPnpSequenceMemory[Call_iProductRecipeNo];

CallStep := 11;


10:
bCallCompleted := TRUE;
CallSelfCheckHR := FALSE;
PreviousProductRecipeCallNo := Call_iProductRecipeNo;
CallStep := 99;

11:

bCallCompleted := TRUE;
CallStep := 99;



99:
;
END_CASE

ACTION XML_ImportExport:
(* XML Import Export Control *)
(*	ARiSubAction					: ARRAY [1..10] OF INT; (* 0-Idle, 1-Import, 2-Export, 3-Clear/Delete 8-Done *)*)


	IF 		ARiSubAction[1] = 1 THEN (*Write from Buffer to Actual Memory*)
				ARDsPnpSequenceMemory[iXMLRecipeNo] := DSV3XML_Recipe.DSProductRecipe;
				ARiSubAction[1] := 8;
(*				IF iHMIRecipeNo = iXMLRecipeNo THEN
					bRecipeLoadPb := TRUE;
				END_IF
*)
	ELSIF	ARiSubAction[1] = 2 THEN (*Read from Actual to Buffer Memory*)
				DSV3XML_Recipe.DSProductRecipe := ARDsPnpSequenceMemory[iXMLRecipeNo];
				ARiSubAction[1] := 8;

	ELSIF	ARiSubAction[1] = 3 THEN (*DELETE Actual Memory*)
				ARDsPnpSequenceMemory := ARDsPnpSequenceMemory_Delete;
				ARiSubAction[1] := 8;
(*				IF iHMIRecipeNo = iXMLRecipeNo THEN
					bRecipeLoadPb := TRUE;
				END_IF
*)
	END_IF
END_ACTION

END_FUNCTION_BLOCK

// ---- FBs/B_JKS_NewFB/FBP-Memory_Sub/fbA21_UpDownPattern.TcPOU
FUNCTION_BLOCK fbA21_UpDownPattern

VAR_INPUT
	bSavePB : BOOL;
	bLoadPB : BOOL;
	bCopyPB : BOOL;
	iCopyToUpDownPatternNo : INT;
END_VAR


VAR_IN_OUT PERSISTENT

	iUpDownPatternNo: INT; (* 10 sets of UpDownPattern *)
	DSinUpDownPatternMemory : DSA21_UpDownPatternMemory;

	Call_iUpDownPatternNo : INT;
	bCallPB: BOOL;

END_VAR
VAR_OUTPUT
	bSaveInd: BOOL;
	bLoadInd: BOOL;
	bCallCompleted : BOOL;
	bInvalidCallUpdownPatternNoHold: BOOL;
	bInvalidCallUpdownPatternNoPulse: BOOL;
	Call_DSUpdownPattern : DSA21_UpDownPatternMemory;

END_VAR
VAR
	SaveIndHr: BOOL;
	LoadIndHr: BOOL;

	SaveTimerDelay: TON;
	LoadTimerDelay: TON;
	SelfCheckTimer: TON;
	bLoadEn: BOOL;
	SelfCheckloopUpdownPattern: BOOL;
	PreviousUpdownPatternNo: INT;

	LoadDF : R_TRIG;
	LoadENDF : R_TRIG;

	SaveDF: R_TRIG;
	CallIntervalTimer: TON;
	CallIntervalDIFU: R_TRIG;

	bCallCompletedHR: BOOL;
	bCallCompletedHRRE: R_TRIG;
	CallCompletedTimer: TON;
	CallSelfCheckTimer : TON;
	CallSelfCheckloop : BOOL;

	CallSelfCheckRE: R_TRIG;
	CallStep: INT;
	CallSelfCheckHR: BOOL;
	bCallPBRE: R_TRIG;

	LoadFL: INT;
	SaveFL: INT;
	PreviousUpdownPatternCallNo: INT;
	CallSFL: INT;
	febInvalidCallUpdownPatternNo: F_TRIG;



	rebInvalidCallUpdownPatternNo: R_TRIG;
	tInvalidCallUpdownPatternNoPulseTimer: TON;
	CopyDF: R_TRIG;
	iMaxMinFL: INT;
END_VAR

VAR PERSISTENT

	ARDsUpdownPatternMemory : ARRAY [1..iArmUpDownPatternArrayQty] OF DSA21_UpDownPatternMemory;
	ARsStorageUpdownPatternDescription: ARRAY [0..iArmUpDownPatternArrayQty] OF STRING(50);


END_VAR

IF iUpDownPatternNo < 1 THEN
iUpDownPatternNo := 1;
END_IF

IF iUpDownPatternNo > iArmUpDownPatternArrayQty THEN
iUpDownPatternNo := iArmUpDownPatternArrayQty;
END_IF


(*Min / Max Control*)
IF DSinUpDownPatternMemory.iZone1SpdProfileNo <= 0 THEN
DSinUpDownPatternMemory.iZone1SpdProfileNo:= 1;
ELSIF DSinUpDownPatternMemory.iZone1SpdProfileNo > iArmSpeedProfileArrayQty THEN
DSinUpDownPatternMemory.iZone1SpdProfileNo:= iArmSpeedProfileArrayQty;
END_IF

IF DSinUpDownPatternMemory.iZone2SpdProfileNo <= 0 THEN
DSinUpDownPatternMemory.iZone2SpdProfileNo:= 1;
ELSIF DSinUpDownPatternMemory.iZone2SpdProfileNo > iArmSpeedProfileArrayQty THEN
DSinUpDownPatternMemory.iZone2SpdProfileNo:= iArmSpeedProfileArrayQty;
END_IF

IF DSinUpDownPatternMemory.iZone3SpdProfileNo <= 0 THEN
DSinUpDownPatternMemory.iZone3SpdProfileNo:= 1;
ELSIF DSinUpDownPatternMemory.iZone3SpdProfileNo > iArmSpeedProfileArrayQty THEN
DSinUpDownPatternMemory.iZone3SpdProfileNo:= iArmSpeedProfileArrayQty;
END_IF

IF DSinUpDownPatternMemory.iZone4SpdProfileNo <= 0 THEN
DSinUpDownPatternMemory.iZone4SpdProfileNo:= 1;
ELSIF DSinUpDownPatternMemory.iZone4SpdProfileNo > iArmSpeedProfileArrayQty THEN
DSinUpDownPatternMemory.iZone4SpdProfileNo:= iArmSpeedProfileArrayQty;
END_IF





(*Load and Save Indicator*)
IF bSavePB THEN
SaveIndHr := TRUE;
END_IF

SaveTimerDelay(IN:=SaveIndHr, PT := T#1s, Q=>, ET=>);
IF SaveTimerDelay.Q THEN
SaveIndHr := FALSE;
END_IF

IF SaveIndHr AND NOT SaveTimerDelay.Q THEN
bSaveInd := TRUE;
ELSE
bSaveInd := FALSE;
END_IF

IF bLoadPB THEN
LoadIndHr := TRUE;
END_IF

LoadTimerDelay(IN:=LoadIndHr, PT := T#1s, Q=>, ET=>);
IF loadtimerdelay.Q THEN
LoadIndHr := FALSE;
END_IF

IF loadIndHr AND NOT LoadTimerDelay.Q THEN
bLoadInd := TRUE;
ELSE
bLoadInd := FALSE;
END_IF

IF iUpDownPatternNo <> PreviousUpdownPatternNo THEN
bLoadEn := TRUE;
ELSE
bLoadEn := FALSE;
END_IF


(* Load Recipe *)

LoadDF(CLK:=bLoadPB,Q=>);
LoadENDF(CLK:=bLoadEn,Q=>);

IF LoadDF.Q OR LoadENDF.Q THEN

DSinUpDownPatternMemory := ARDsUpdownPatternMemory[iUpDownPatternNo];
PreviousUpdownPatternNo := iUpDownPatternNo  ;

END_IF


(* Save Recipe *)

SaveDF(CLK:=bSavePB,Q=>);

IF SaveDF.Q THEN

ARDsUpdownPatternMemory[iUpDownPatternNo] := DSinUpDownPatternMemory;
ARsStorageUpdownPatternDescription[iUpDownPatternNo] := DSinUpDownPatternMemory.sDescription;

END_IF


(*Copy Recipe*)

CopyDF(CLK:=bCopyPB,Q=>);

IF CopyDF.Q THEN

ARDsUpdownPatternMemory[iCopyToUpDownPatternNo] := ARDsUpdownPatternMemory[iUpDownPatternNo];
ARsStorageUpdownPatternDescription[iCopyToUpDownPatternNo] := ARDsUpdownPatternMemory[iUpDownPatternNo].sDescription;

END_IF





(* Call Recipe *)
(* ---- Call Recipe Complete Flag ---*)


IF NOT bCallPB THEN
bCallCompleted := FALSE;
END_IF

bCallPBRE(CLK:=bCallPB , Q=> );

IF (Call_iUpDownPatternNo <= 0 OR Call_iUpDownPatternNo > iArmUpDownPatternArrayQty) AND bCallPB THEN
bInvalidCallUpdownPatternNoHold := TRUE;
ELSE
bInvalidCallUpdownPatternNoHold := FALSE;
END_IF


